KUKA KRL program: MyProgram_002().src

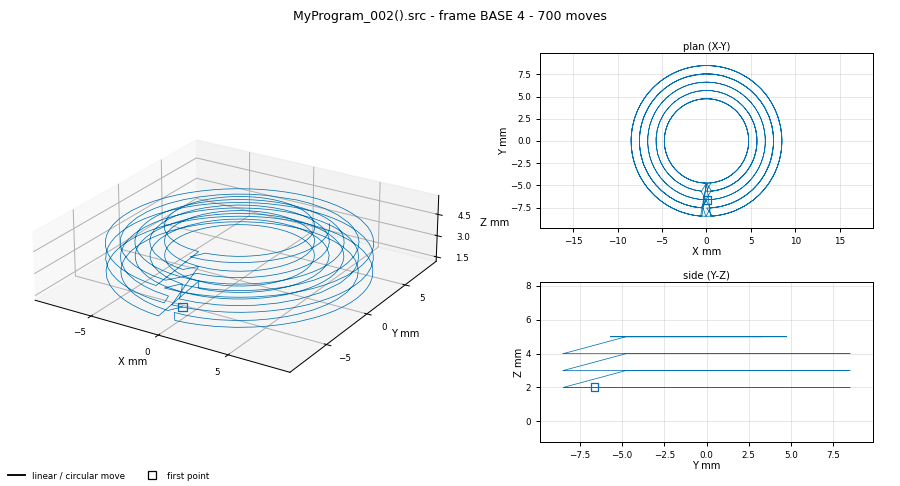
[picture p0: tool path of MyProgram_002().src in frame BASE 4, 700 of 700 moves have a stored position in this frame; points joined in program order, loops and branches not executed]
&ACCESS RVP
&REL 1
&PARAM TEMPLATE = C:\KRC\Roboter\Template\vorgabe
&PARAM EDITMASK = *
DEF MyProgram_002()
; ---- Setting reference (Base) ----
$BASE = BASE_DATA[4]

; --------------------------
; ---- Setting tool (TCP) ----
$TOOL = TOOL_DATA[3]
; --------------------------

$VEL.CP = VEL_APROX_PRINT
Startdeposition()
$VEL.CP = VEL_PRINT
LIN {X 0.0178,Y -6.6224,Z 2,A -3.1111,B 0,C 0,E1 0.1598,E2 90.0714} C_DIS
Enddeposition()
LIN {X 0.0178,Y -6.6224,Z 2,A -3.1111,B 0,C 0,E1 0.1598,E2 90.0714} C_DIS
Startdeposition()
$VEL.CP = VEL_PRINT
LIN {X -0.4593,Y -7.5388,Z 2,A -3.167,B 0,C 0,E1 0.1598,E2 90.0708} C_DIS
LIN {X -1.4599,Y -7.4149,Z 2,A -3.199,B 0,C 0,E1 0.1598,E2 90.0713} C_DIS
LIN {X -2.4674,Y -7.1388,Z 2,A -3.2242,B 0,C 0,E1 0.1598,E2 90.0713} C_DIS
LIN {X -3.4306,Y -6.7344,Z 2,A -3.2424,B 0,C 0,E1 0.1598,E2 90.0711} C_DIS
LIN {X -4.2642,Y -6.2384,Z 2,A -3.252,B 0,C 0,E1 0.1598,E2 90.0711} C_DIS
LIN {X -5.1322,Y -5.543,Z 2,A -3.2544,B 0,C 0,E1 0.1598,E2 90.071} C_DIS
LIN {X -5.6941,Y -4.9627,Z 2,A -3.2507,B 0,C 0,E1 0.1598,E2 90.071} C_DIS
LIN {X -6.1903,Y -4.3255,Z 2,A -3.242,B 0,C 0,E1 0.1598,E2 90.071} C_DIS
LIN {X -6.7788,Y -3.3392,Z 2,A -3.2218,B 0,C 0,E1 0.1598,E2 90.0708} C_DIS
LIN {X -7.1266,Y -2.5145,Z 2,A -3.2,B 0,C 0,E1 0.1598,E2 90.0708} C_DIS
LIN {X -7.4318,Y -1.3786,Z 2,A -3.1631,B 0,C 0,E1 0.1598,E2 90.0708} C_DIS
LIN {X -7.5532,Y -0.2507,Z 2,A -3.1202,B 0,C 0,E1 0.1598,E2 90.0708} C_DIS
LIN {X -7.507,Y 0.8388,Z 2,A -3.0728,B 0,C 0,E1 0.1598,E2 90.0709} C_DIS
LIN {X -7.3592,Y 1.6986,Z 2,A -3.0313,B 0,C 0,E1 0.1598,E2 90.0712} C_DIS
LIN {X -7.0429,Y 2.7423,Z 2,A -2.9756,B 0,C 0,E1 0.1598,E2 90.071} C_DIS
LIN {X -6.514,Y 3.8232,Z 2,A -2.9107,B 0,C 0,E1 0.1598,E2 90.0711} C_DIS
LIN {X -6.0604,Y 4.5077,Z 2,A -2.8655,B 0,C 0,E1 0.1598,E2 90.0715} C_DIS
LIN {X -5.5355,Y 5.1393,Z 2,A -2.8197,B 0,C 0,E1 0.1598,E2 90.0716} C_DIS
LIN {X -4.7193,Y 5.9031,Z 2,A -2.7574,B 0,C 0,E1 0.1598,E2 90.0716} C_DIS
LIN {X -3.7399,Y 6.5671,Z 2,A -2.6934,B 0,C 0,E1 0.1598,E2 90.0718} C_DIS
LIN {X -2.7889,Y 7.019,Z 2,A -2.6394,B 0,C 0,E1 0.1598,E2 90.072} C_DIS
LIN {X -1.9903,Y 7.2868,Z 2,A -2.5987,B 0,C 0,E1 0.1598,E2 90.072} C_DIS
LIN {X -1.1667,Y 7.463,Z 2,A -2.5609,B 0,C 0,E1 0.1598,E2 90.0721} C_DIS
LIN {X -0.118,Y 7.5562,Z 2,A -2.5182,B 0,C 0,E1 0.1598,E2 90.0722} C_DIS
LIN {X 1.0472,Y 7.4801,Z 2,A -2.4784,B 0,C 0,E1 0.1598,E2 90.0722} C_DIS
LIN {X 1.8826,Y 7.3157,Z 2,A -2.4545,B 0,C 0,E1 0.1598,E2 90.0722} C_DIS
LIN {X 2.9847,Y 6.9422,Z 2,A -2.4295,B 0,C 0,E1 0.1598,E2 90.0722} C_DIS
LIN {X 3.8476,Y 6.5002,Z 2,A -2.4163,B 0,C 0,E1 0.1598,E2 90.0722} C_DIS
LIN {X 4.7671,Y 5.8658,Z 2,A -2.409,B 0,C 0,E1 0.1598,E2 90.0722} C_DIS
LIN {X 5.5879,Y 5.0811,Z 2,A -2.4118,B 0,C 0,E1 0.1598,E2 90.072} C_DIS
LIN {X 6.1162,Y 4.4317,Z 2,A -2.4199,B 0,C 0,E1 0.1598,E2 90.072} C_DIS
LIN {X 6.5685,Y 3.7273,Z 2,A -2.433,B 0,C 0,E1 0.1598,E2 90.072} C_DIS
LIN {X 7.0263,Y 2.7862,Z 2,A -2.4557,B 0,C 0,E1 0.1598,E2 90.0717} C_DIS
LIN {X 7.3641,Y 1.6742,Z 2,A -2.4903,B 0,C 0,E1 0.1598,E2 90.0715} C_DIS
LIN {X 7.5359,Y 0.5664,Z 2,A -2.5309,B 0,C 0,E1 0.1598,E2 90.0715} C_DIS
LIN {X 7.5261,Y -0.6981,Z 2,A -2.5848,B 0,C 0,E1 0.1598,E2 90.0713} C_DIS
LIN {X 7.3558,Y -1.7123,Z 2,A -2.6343,B 0,C 0,E1 0.1598,E2 90.0715} C_DIS
LIN {X 7.0595,Y -2.6971,Z 2,A -2.6869,B 0,C 0,E1 0.1598,E2 90.0714} C_DIS
LIN {X 6.5954,Y -3.6789,Z 2,A -2.7457,B 0,C 0,E1 0.1598,E2 90.0714} C_DIS
LIN {X 6.1284,Y -4.4233,Z 2,A -2.7946,B 0,C 0,E1 0.1598,E2 90.0715} C_DIS
LIN {X 5.3883,Y -5.2916,Z 2,A -2.8585,B 0,C 0,E1 0.1598,E2 90.0714} C_DIS
LIN {X 4.762,Y -5.8618,Z 2,A -2.9059,B 0,C 0,E1 0.1598,E2 90.0715} C_DIS
LIN {X 3.8982,Y -6.4739,Z 2,A -2.9635,B 0,C 0,E1 0.1598,E2 90.0715} C_DIS
LIN {X 2.7755,Y -7.0305,Z 2,A -3.0283,B 0,C 0,E1 0.1598,E2 90.0714} C_DIS
LIN {X 1.7367,Y -7.3513,Z 2,A -3.0801,B 0,C 0,E1 0.1598,E2 90.0714} C_DIS
LIN {X 0.7907,Y -7.5156,Z 2,A -3.1218,B 0,C 0,E1 0.1598,E2 90.0714} C_DIS
LIN {X 0.024,Y -7.5549,Z 2,A -3.1516,B 0,C 0,E1 0.1598,E2 90.0714} C_DIS
Enddeposition()
LIN {X 0.024,Y -7.5549,Z 2,A -3.1516,B 0,C 0,E1 0.1598,E2 90.0714} C_DIS
Startdeposition()
$VEL.CP = VEL_PRINT
LIN {X 0.6615,Y -8.4625,Z 2,A -3.1663,B 0,C 0,E1 0.1598,E2 90.0708} C_DIS
LIN {X 1.4734,Y -8.3591,Z 2,A -3.1326,B 0,C 0,E1 0.1598,E2 90.0714} C_DIS
LIN {X 2.2716,Y -8.1784,Z 2,A -3.0957,B 0,C 0,E1 0.1598,E2 90.0714} C_DIS
LIN {X 3.2398,Y -7.8482,Z 2,A -3.0462,B 0,C 0,E1 0.1598,E2 90.0714} C_DIS
LIN {X 4.3203,Y -7.3105,Z 2,A -2.9837,B 0,C 0,E1 0.1598,E2 90.0714} C_DIS
LIN {X 5.1942,Y -6.7139,Z 2,A -2.9263,B 0,C 0,E1 0.1598,E2 90.0715} C_DIS
LIN {X 5.8372,Y -6.1633,Z 2,A -2.8794,B 0,C 0,E1 0.1598,E2 90.0715} C_DIS
LIN {X 6.4222,Y -5.5514,Z 2,A -2.8319,B 0,C 0,E1 0.1598,E2 90.0716} C_DIS
LIN {X 7.0647,Y -4.7107,Z 2,A -2.7724,B 0,C 0,E1 0.1598,E2 90.0715} C_DIS
LIN {X 7.6515,Y -3.6709,Z 2,A -2.7066,B 0,C 0,E1 0.1598,E2 90.0715} C_DIS
LIN {X 7.9615,Y -2.9397,Z 2,A -2.6644,B 0,C 0,E1 0.1598,E2 90.0717} C_DIS
LIN {X 8.2023,Y -2.1829,Z 2,A -2.6234,B 0,C 0,E1 0.1598,E2 90.0717} C_DIS
LIN {X 8.3716,Y -1.4069,Z 2,A -2.5843,B 0,C 0,E1 0.1598,E2 90.0718} C_DIS
LIN {X 8.4662,Y -0.6183,Z 2,A -2.5473,B 0,C 0,E1 0.1598,E2 90.0718} C_DIS
LIN {X 8.4863,Y 0.1757,Z 2,A -2.5129,B 0,C 0,E1 0.1598,E2 90.0718} C_DIS
LIN {X 8.4313,Y 0.968,Z 2,A -2.4813,B 0,C 0,E1 0.1598,E2 90.0719} C_DIS
LIN {X 8.3033,Y 1.7517,Z 2,A -2.4527,B 0,C 0,E1 0.1598,E2 90.0719} C_DIS
LIN {X 8.1033,Y 2.5202,Z 2,A -2.4275,B 0,C 0,E1 0.1598,E2 90.0719} C_DIS
LIN {X 7.7584,Y 3.4511,Z 2,A -2.4005,B 0,C 0,E1 0.1598,E2 90.0719} C_DIS
LIN {X 7.165,Y 4.5511,Z 2,A -2.3757,B 0,C 0,E1 0.1598,E2 90.0717} C_DIS
LIN {X 6.6849,Y 5.2318,Z 2,A -2.365,B 0,C 0,E1 0.1598,E2 90.0721} C_DIS
LIN {X 6.1405,Y 5.8622,Z 2,A -2.3584,B 0,C 0,E1 0.1598,E2 90.0721} C_DIS
LIN {X 5.3784,Y 6.5716,Z 2,A -2.3564,B 0,C 0,E1 0.1598,E2 90.0721} C_DIS
LIN {X 4.6112,Y 7.1308,Z 2,A -2.3613,B 0,C 0,E1 0.1598,E2 90.0722} C_DIS
LIN {X 3.6186,Y 7.681,Z 2,A -2.3747,B 0,C 0,E1 0.1598,E2 90.0722} C_DIS
LIN {X 2.6506,Y 8.0636,Z 2,A -2.3944,B 0,C 0,E1 0.1598,E2 90.0722} C_DIS
LIN {X 1.8478,Y 8.2847,Z 2,A -2.4147,B 0,C 0,E1 0.1598,E2 90.0723} C_DIS
LIN {X 1.0272,Y 8.4264,Z 2,A -2.4391,B 0,C 0,E1 0.1598,E2 90.0723} C_DIS
LIN {X 0.1966,Y 8.4864,Z 2,A -2.4673,B 0,C 0,E1 0.1598,E2 90.0723} C_DIS
LIN {X -0.6357,Y 8.465,Z 2,A -2.4989,B 0,C 0,E1 0.1598,E2 90.0723} C_DIS
LIN {X -1.4619,Y 8.3604,Z 2,A -2.5338,B 0,C 0,E1 0.1598,E2 90.0722} C_DIS
LIN {X -2.2742,Y 8.1774,Z 2,A -2.5715,B 0,C 0,E1 0.1598,E2 90.0722} C_DIS
LIN {X -3.0645,Y 7.9151,Z 2,A -2.6117,B 0,C 0,E1 0.1598,E2 90.0721} C_DIS
LIN {X -3.8254,Y 7.5768,Z 2,A -2.654,B 0,C 0,E1 0.1598,E2 90.072} C_DIS
LIN {X -4.5496,Y 7.1657,Z 2,A -2.698,B 0,C 0,E1 0.1598,E2 90.0719} C_DIS
LIN {X -5.2302,Y 6.6859,Z 2,A -2.7433,B 0,C 0,E1 0.1598,E2 90.0719} C_DIS
LIN {X -5.8601,Y 6.1413,Z 2,A -2.7894,B 0,C 0,E1 0.1598,E2 90.0717} C_DIS
LIN {X -6.4342,Y 5.5382,Z 2,A -2.8359,B 0,C 0,E1 0.1598,E2 90.0717} C_DIS
LIN {X -6.9449,Y 4.8805,Z 2,A -2.8823,B 0,C 0,E1 0.1598,E2 90.0715} C_DIS
LIN {X -7.3896,Y 4.1765,Z 2,A -2.9282,B 0,C 0,E1 0.1598,E2 90.0715} C_DIS
LIN {X -7.763,Y 3.4322,Z 2,A -2.9732,B 0,C 0,E1 0.1598,E2 90.0713} C_DIS
LIN {X -8.062,Y 2.655,Z 2,A -3.0168,B 0,C 0,E1 0.1598,E2 90.0713} C_DIS
LIN {X -8.2835,Y 1.8523,Z 2,A -3.0587,B 0,C 0,E1 0.1598,E2 90.0712} C_DIS
LIN {X -8.4257,Y 1.0318,Z 2,A -3.0984,B 0,C 0,E1 0.1598,E2 90.0712} C_DIS
LIN {X -8.4869,Y 0.2014,Z 2,A -3.1355,B 0,C 0,E1 0.1598,E2 90.071} C_DIS
LIN {X -8.4655,Y -0.631,Z 2,A -3.1697,B 0,C 0,E1 0.1598,E2 90.071} C_DIS
LIN {X -8.3623,Y -1.4573,Z 2,A -3.2006,B 0,C 0,E1 0.1598,E2 90.071} C_DIS
LIN {X -8.1789,Y -2.2696,Z 2,A -3.2281,B 0,C 0,E1 0.1598,E2 90.071} C_DIS
LIN {X -7.9171,Y -3.0601,Z 2,A -3.2517,B 0,C 0,E1 0.1598,E2 90.071} C_DIS
LIN {X -7.5792,Y -3.8212,Z 2,A -3.2713,B 0,C 0,E1 0.1598,E2 90.071} C_DIS
LIN {X -7.0571,Y -4.7217,Z 2,A -3.2899,B 0,C 0,E1 0.1598,E2 90.0707} C_DIS
LIN {X -6.3174,Y -5.6752,Z 2,A -3.3028,B 0,C 0,E1 0.1598,E2 90.0707} C_DIS
LIN {X -5.5366,Y -6.4363,Z 2,A -3.3065,B 0,C 0,E1 0.1598,E2 90.0709} C_DIS
LIN {X -4.7817,Y -7.0119,Z 2,A -3.3032,B 0,C 0,E1 0.1598,E2 90.071} C_DIS
LIN {X -4.136,Y -7.4117,Z 2,A -3.2965,B 0,C 0,E1 0.1598,E2 90.071} C_DIS
LIN {X -3.4569,Y -7.7519,Z 2,A -3.286,B 0,C 0,E1 0.1598,E2 90.0711} C_DIS
LIN {X -2.7497,Y -8.0287,Z 2,A -3.2717,B 0,C 0,E1 0.1598,E2 90.0711} C_DIS
LIN {X -2.021,Y -8.2422,Z 2,A -3.2541,B 0,C 0,E1 0.1598,E2 90.0712} C_DIS
LIN {X -1.2762,Y -8.3903,Z 2,A -3.233,B 0,C 0,E1 0.1598,E2 90.0712} C_DIS
LIN {X -0.5212,Y -8.4723,Z 2,A -3.2088,B 0,C 0,E1 0.1598,E2 90.0712} C_DIS
LIN {X -0.5212,Y -8.4723,Z 2,A -3.2088,B 0,C 0,E1 0.1598,E2 90.0712} C_DIS
Enddeposition()
LIN {X 0.0002,Y -4.757,Z 3,A -3.0171,B 0,C 0,E1 0.1598,E2 90.0603} C_DIS
Startdeposition()
$VEL.CP = VEL_PRINT
LIN {X 0.0002,Y -4.757,Z 3,A -3.0228,B 0,C 0,E1 0.1598,E2 90.066} C_DIS
LIN {X -0.6823,Y -4.7037,Z 3,A -3.0504,B 0,C 0,E1 0.1598,E2 90.0709} C_DIS
LIN {X -1.2189,Y -4.5944,Z 3,A -3.0661,B 0,C 0,E1 0.1598,E2 90.0714} C_DIS
LIN {X -1.7393,Y -4.4237,Z 3,A -3.078,B 0,C 0,E1 0.1598,E2 90.0714} C_DIS
LIN {X -2.2363,Y -4.1936,Z 3,A -3.0865,B 0,C 0,E1 0.1598,E2 90.0714} C_DIS
LIN {X -2.7046,Y -3.9096,Z 3,A -3.0917,B 0,C 0,E1 0.1598,E2 90.0714} C_DIS
LIN {X -3.1363,Y -3.5726,Z 3,A -3.0933,B 0,C 0,E1 0.1598,E2 90.0714} C_DIS
LIN {X -3.5248,Y -3.1869,Z 3,A -3.0913,B 0,C 0,E1 0.1598,E2 90.0714} C_DIS
LIN {X -3.868,Y -2.7601,Z 3,A -3.0859,B 0,C 0,E1 0.1598,E2 90.0714} C_DIS
LIN {X -4.1606,Y -2.297,Z 3,A -3.0771,B 0,C 0,E1 0.1598,E2 90.0714} C_DIS
LIN {X -4.3949,Y -1.8023,Z 3,A -3.0649,B 0,C 0,E1 0.1598,E2 90.0714} C_DIS
LIN {X -4.5762,Y -1.2855,Z 3,A -3.0497,B 0,C 0,E1 0.1598,E2 90.0714} C_DIS
LIN {X -4.6927,Y -0.7504,Z 3,A -3.0315,B 0,C 0,E1 0.1598,E2 90.0714} C_DIS
LIN {X -4.7468,Y -0.2055,Z 3,A -3.0105,B 0,C 0,E1 0.1598,E2 90.0714} C_DIS
LIN {X -4.7423,Y 0.3421,Z 3,A -2.9873,B 0,C 0,E1 0.1598,E2 90.0714} C_DIS
LIN {X -4.6683,Y 0.8848,Z 3,A -2.9617,B 0,C 0,E1 0.1598,E2 90.0714} C_DIS
LIN {X -4.5367,Y 1.4164,Z 3,A -2.9345,B 0,C 0,E1 0.1598,E2 90.0715} C_DIS
LIN {X -4.3445,Y 1.9292,Z 3,A -2.9058,B 0,C 0,E1 0.1598,E2 90.0715} C_DIS
LIN {X -4.0931,Y 2.4158,Z 3,A -2.8761,B 0,C 0,E1 0.1598,E2 90.0716} C_DIS
LIN {X -3.7885,Y 2.8709,Z 3,A -2.8457,B 0,C 0,E1 0.1598,E2 90.0716} C_DIS
LIN {X -3.434,Y 3.2883,Z 3,A -2.8151,B 0,C 0,E1 0.1598,E2 90.0717} C_DIS
LIN {X -3.0321,Y 3.6604,Z 3,A -2.7846,B 0,C 0,E1 0.1598,E2 90.0717} C_DIS
LIN {X -2.5909,Y 3.9849,Z 3,A -2.7547,B 0,C 0,E1 0.1598,E2 90.0719} C_DIS
LIN {X -2.1155,Y 4.2567,Z 3,A -2.7257,B 0,C 0,E1 0.1598,E2 90.0719} C_DIS
LIN {X -1.6115,Y 4.4711,Z 3,A -2.6981,B 0,C 0,E1 0.1598,E2 90.0719} C_DIS
LIN {X -1.0866,Y 4.6274,Z 3,A -2.6722,B 0,C 0,E1 0.1598,E2 90.072} C_DIS
LIN {X -0.5471,Y 4.7215,Z 3,A -2.6483,B 0,C 0,E1 0.1598,E2 90.072} C_DIS
LIN {X -0.0003,Y 4.753,Z 3,A -2.6268,B 0,C 0,E1 0.1598,E2 90.072} C_DIS
LIN {X 0.5465,Y 4.7225,Z 3,A -2.608,B 0,C 0,E1 0.1598,E2 90.072} C_DIS
LIN {X 1.0858,Y 4.6272,Z 3,A -2.5921,B 0,C 0,E1 0.1598,E2 90.0721} C_DIS
LIN {X 1.6101,Y 4.469,Z 3,A -2.5794,B 0,C 0,E1 0.1598,E2 90.0721} C_DIS
LIN {X 2.1146,Y 4.2565,Z 3,A -2.5698,B 0,C 0,E1 0.1598,E2 90.0721} C_DIS
LIN {X 2.5892,Y 3.9833,Z 3,A -2.5638,B 0,C 0,E1 0.1598,E2 90.0721} C_DIS
LIN {X 3.0305,Y 3.6591,Z 3,A -2.5612,B 0,C 0,E1 0.1598,E2 90.0721} C_DIS
LIN {X 3.433,Y 3.2877,Z 3,A -2.5621,B 0,C 0,E1 0.1598,E2 90.0721} C_DIS
LIN {X 3.7883,Y 2.8711,Z 3,A -2.5666,B 0,C 0,E1 0.1598,E2 90.0721} C_DIS
LIN {X 4.0916,Y 2.4151,Z 3,A -2.5747,B 0,C 0,E1 0.1598,E2 90.0721} C_DIS
LIN {X 4.3444,Y 1.9293,Z 3,A -2.5859,B 0,C 0,E1 0.1598,E2 90.072} C_DIS
LIN {X 4.5367,Y 1.4166,Z 3,A -2.6005,B 0,C 0,E1 0.1598,E2 90.072} C_DIS
LIN {X 4.6699,Y 0.8853,Z 3,A -2.6181,B 0,C 0,E1 0.1598,E2 90.072} C_DIS
LIN {X 4.7423,Y 0.3424,Z 3,A -2.6384,B 0,C 0,E1 0.1598,E2 90.0719} C_DIS
LIN {X 4.7478,Y -0.2053,Z 3,A -2.6614,B 0,C 0,E1 0.1598,E2 90.0719} C_DIS
LIN {X 4.6939,Y -0.7501,Z 3,A -2.6864,B 0,C 0,E1 0.1598,E2 90.0719} C_DIS
LIN {X 4.5744,Y -1.2846,Z 3,A -2.7135,B 0,C 0,E1 0.1598,E2 90.0719} C_DIS
LIN {X 4.3976,Y -1.8028,Z 3,A -2.7419,B 0,C 0,E1 0.1598,E2 90.0718} C_DIS
LIN {X 4.1613,Y -2.2969,Z 3,A -2.7716,B 0,C 0,E1 0.1598,E2 90.0718} C_DIS
LIN {X 3.87,Y -2.7606,Z 3,A -2.8019,B 0,C 0,E1 0.1598,E2 90.0718} C_DIS
LIN {X 3.5258,Y -3.1866,Z 3,A -2.8326,B 0,C 0,E1 0.1598,E2 90.0718} C_DIS
LIN {X 3.1365,Y -3.5719,Z 3,A -2.8633,B 0,C 0,E1 0.1598,E2 90.0717} C_DIS
LIN {X 2.7044,Y -3.9081,Z 3,A -2.8934,B 0,C 0,E1 0.1598,E2 90.0717} C_DIS
LIN {X 2.2361,Y -4.1922,Z 3,A -2.9226,B 0,C 0,E1 0.1598,E2 90.0717} C_DIS
LIN {X 1.7398,Y -4.4234,Z 3,A -2.9507,B 0,C 0,E1 0.1598,E2 90.0717} C_DIS
LIN {X 1.2188,Y -4.5918,Z 3,A -2.9769,B 0,C 0,E1 0.1598,E2 90.0716} C_DIS
LIN {X 0.6827,Y -4.7037,Z 3,A -3.0014,B 0,C 0,E1 0.1598,E2 90.0716} C_DIS
LIN {X 0.0002,Y -4.757,Z 3,A -3.0287,B 0,C 0,E1 0.1598,E2 90.0716} C_DIS
Enddeposition()
LIN {X 0.0002,Y -4.757,Z 3,A -3.0287,B 0,C 0,E1 0.1598,E2 90.0716} C_DIS
Startdeposition()
$VEL.CP = VEL_PRINT
LIN {X 0.5659,Y -5.6547,Z 3,A -3.0454,B 0,C 0,E1 0.1598,E2 90.071} C_DIS
LIN {X 1.3547,Y -5.5195,Z 3,A -3.0113,B 0,C 0,E1 0.1598,E2 90.0715} C_DIS
LIN {X 2.1165,Y -5.2741,Z 3,A -2.9729,B 0,C 0,E1 0.1598,E2 90.0715} C_DIS
LIN {X 2.8372,Y -4.9256,Z 3,A -2.9317,B 0,C 0,E1 0.1598,E2 90.0716} C_DIS
LIN {X 3.5009,Y -4.4782,Z 3,A -2.8883,B 0,C 0,E1 0.1598,E2 90.0716} C_DIS
LIN {X 4.0958,Y -3.9425,Z 3,A -2.8437,B 0,C 0,E1 0.1598,E2 90.0716} C_DIS
LIN {X 4.6092,Y -3.3282,Z 3,A -2.7988,B 0,C 0,E1 0.1598,E2 90.0716} C_DIS
LIN {X 5.0292,Y -2.6467,Z 3,A -2.7544,B 0,C 0,E1 0.1598,E2 90.0716} C_DIS
LIN {X 5.3532,Y -1.9147,Z 3,A -2.7115,B 0,C 0,E1 0.1598,E2 90.0716} C_DIS
LIN {X 5.5679,Y -1.1434,Z 3,A -2.6708,B 0,C 0,E1 0.1598,E2 90.0716} C_DIS
LIN {X 5.6733,Y -0.35,Z 3,A -2.6333,B 0,C 0,E1 0.1598,E2 90.0717} C_DIS
LIN {X 5.6642,Y 0.4503,Z 3,A -2.5997,B 0,C 0,E1 0.1598,E2 90.0717} C_DIS
LIN {X 5.5458,Y 1.2418,Z 3,A -2.5706,B 0,C 0,E1 0.1598,E2 90.0717} C_DIS
LIN {X 5.3166,Y 2.0087,Z 3,A -2.5465,B 0,C 0,E1 0.1598,E2 90.0718} C_DIS
LIN {X 4.8879,Y 2.9128,Z 3,A -2.5239,B 0,C 0,E1 0.1598,E2 90.0717} C_DIS
LIN {X 4.2073,Y 3.8229,Z 3,A -2.5105,B 0,C 0,E1 0.1598,E2 90.0717} C_DIS
LIN {X 3.615,Y 4.3886,Z 3,A -2.5087,B 0,C 0,E1 0.1598,E2 90.072} C_DIS
LIN {X 2.9467,Y 4.8621,Z 3,A -2.5134,B 0,C 0,E1 0.1598,E2 90.072} C_DIS
LIN {X 2.2169,Y 5.2338,Z 3,A -2.5246,B 0,C 0,E1 0.1598,E2 90.0721} C_DIS
LIN {X 1.4422,Y 5.4988,Z 3,A -2.5421,B 0,C 0,E1 0.1598,E2 90.0721} C_DIS
LIN {X 0.6371,Y 5.6481,Z 3,A -2.5655,B 0,C 0,E1 0.1598,E2 90.0721} C_DIS
LIN {X -0.181,Y 5.68,Z 3,A -2.5944,B 0,C 0,E1 0.1598,E2 90.0721} C_DIS
LIN {X -0.9954,Y 5.5962,Z 3,A -2.6279,B 0,C 0,E1 0.1598,E2 90.0721} C_DIS
LIN {X -1.7885,Y 5.3936,Z 3,A -2.6657,B 0,C 0,E1 0.1598,E2 90.0721} C_DIS
LIN {X -2.9131,Y 4.8877,Z 3,A -2.7284,B 0,C 0,E1 0.1598,E2 90.0718} C_DIS
LIN {X -3.6482,Y 4.3607,Z 3,A -2.7777,B 0,C 0,E1 0.1598,E2 90.0718} C_DIS
LIN {X -4.2376,Y 3.7904,Z 3,A -2.8234,B 0,C 0,E1 0.1598,E2 90.0716} C_DIS
LIN {X -4.7386,Y 3.1413,Z 3,A -2.8691,B 0,C 0,E1 0.1598,E2 90.0716} C_DIS
LIN {X -5.2815,Y 2.117,Z 3,A -2.9319,B 0,C 0,E1 0.1598,E2 90.0712} C_DIS
LIN {X -5.5389,Y 1.2778,Z 3,A -2.9769,B 0,C 0,E1 0.1598,E2 90.0712} C_DIS
LIN {X -5.6863,Y 0.2165,Z 3,A -3.0267,B 0,C 0,E1 0.1598,E2 90.071} C_DIS
LIN {X -5.6319,Y -0.7558,Z 3,A -3.0658,B 0,C 0,E1 0.1598,E2 90.071} C_DIS
LIN {X -5.4764,Y -1.5191,Z 3,A -3.0923,B 0,C 0,E1 0.1598,E2 90.0711} C_DIS
LIN {X -5.2196,Y -2.2546,Z 3,A -3.1139,B 0,C 0,E1 0.1598,E2 90.0711} C_DIS
LIN {X -4.8609,Y -2.9464,Z 3,A -3.1299,B 0,C 0,E1 0.1598,E2 90.0711} C_DIS
LIN {X -4.4131,Y -3.5841,Z 3,A -3.1404,B 0,C 0,E1 0.1598,E2 90.0711} C_DIS
LIN {X -3.6555,Y -4.3598,Z 3,A -3.1452,B 0,C 0,E1 0.1598,E2 90.0711} C_DIS
LIN {X -2.8468,Y -4.9172,Z 3,A -3.1391,B 0,C 0,E1 0.1598,E2 90.0712} C_DIS
LIN {X -2.1425,Y -5.2653,Z 3,A -3.1281,B 0,C 0,E1 0.1598,E2 90.0713} C_DIS
LIN {X -1.3959,Y -5.5111,Z 3,A -3.1111,B 0,C 0,E1 0.1598,E2 90.0713} C_DIS
LIN {X -0.6227,Y -5.6519,Z 3,A -3.0887,B 0,C 0,E1 0.1598,E2 90.0714} C_DIS
LIN {X -0.6227,Y -5.6519,Z 3,A -3.0887,B 0,C 0,E1 0.1598,E2 90.0714} C_DIS
Enddeposition()
LIN {X -0.0547,Y -6.6238,Z 3,A -3.1079,B 0,C 0,E1 0.1598,E2 90.0703} C_DIS
Startdeposition()
$VEL.CP = VEL_PRINT
LIN {X -0.9403,Y -6.5528,Z 3,A -3.1385,B 0,C 0,E1 0.1598,E2 90.0713} C_DIS
LIN {X -1.6368,Y -6.4121,Z 3,A -3.1582,B 0,C 0,E1 0.1598,E2 90.0713} C_DIS
LIN {X -2.3151,Y -6.2004,Z 3,A -3.1741,B 0,C 0,E1 0.1598,E2 90.0713} C_DIS
LIN {X -2.9667,Y -5.9167,Z 3,A -3.186,B 0,C 0,E1 0.1598,E2 90.0713} C_DIS
LIN {X -3.5839,Y -5.5645,Z 3,A -3.1938,B 0,C 0,E1 0.1598,E2 90.0713} C_DIS
LIN {X -4.1606,Y -5.1494,Z 3,A -3.1974,B 0,C 0,E1 0.1598,E2 90.0713} C_DIS
LIN {X -4.6878,Y -4.6728,Z 3,A -3.1966,B 0,C 0,E1 0.1598,E2 90.0712} C_DIS
LIN {X -5.1627,Y -4.1443,Z 3,A -3.1917,B 0,C 0,E1 0.1598,E2 90.0712} C_DIS
LIN {X -5.5767,Y -3.5667,Z 3,A -3.1826,B 0,C 0,E1 0.1598,E2 90.0712} C_DIS
LIN {X -5.9281,Y -2.9489,Z 3,A -3.1694,B 0,C 0,E1 0.1598,E2 90.0712} C_DIS
LIN {X -6.2073,Y -2.2953,Z 3,A -3.1521,B 0,C 0,E1 0.1598,E2 90.0712} C_DIS
LIN {X -6.4184,Y -1.6168,Z 3,A -3.1313,B 0,C 0,E1 0.1598,E2 90.0712} C_DIS
LIN {X -6.555,Y -0.9194,Z 3,A -3.107,B 0,C 0,E1 0.1598,E2 90.0712} C_DIS
LIN {X -6.6162,Y -0.2115,Z 3,A -3.0794,B 0,C 0,E1 0.1598,E2 90.0712} C_DIS
LIN {X -6.6006,Y 0.499,Z 3,A -3.049,B 0,C 0,E1 0.1598,E2 90.0712} C_DIS
LIN {X -6.5101,Y 1.2038,Z 3,A -3.016,B 0,C 0,E1 0.1598,E2 90.0713} C_DIS
LIN {X -6.344,Y 1.8948,Z 3,A -2.9808,B 0,C 0,E1 0.1598,E2 90.0713} C_DIS
LIN {X -6.1053,Y 2.5642,Z 3,A -2.9439,B 0,C 0,E1 0.1598,E2 90.0714} C_DIS
LIN {X -5.7956,Y 3.2039,Z 3,A -2.9056,B 0,C 0,E1 0.1598,E2 90.0714} C_DIS
LIN {X -5.4182,Y 3.8062,Z 3,A -2.8664,B 0,C 0,E1 0.1598,E2 90.0716} C_DIS
LIN {X -4.9762,Y 4.3628,Z 3,A -2.8267,B 0,C 0,E1 0.1598,E2 90.0716} C_DIS
LIN {X -4.4816,Y 4.8729,Z 3,A -2.787,B 0,C 0,E1 0.1598,E2 90.0717} C_DIS
LIN {X -3.9323,Y 5.3238,Z 3,A -2.7478,B 0,C 0,E1 0.1598,E2 90.0718} C_DIS
LIN {X -3.3399,Y 5.7162,Z 3,A -2.7094,B 0,C 0,E1 0.1598,E2 90.0718} C_DIS
LIN {X -2.7081,Y 6.0415,Z 3,A -2.6725,B 0,C 0,E1 0.1598,E2 90.072} C_DIS
LIN {X -2.0452,Y 6.2975,Z 3,A -2.6372,B 0,C 0,E1 0.1598,E2 90.072} C_DIS
LIN {X -1.3586,Y 6.4813,Z 3,A -2.6042,B 0,C 0,E1 0.1598,E2 90.072} C_DIS
LIN {X -0.656,Y 6.5872,Z 3,A -2.5738,B 0,C 0,E1 0.1598,E2 90.0721} C_DIS
LIN {X 0.0541,Y 6.6202,Z 3,A -2.5462,B 0,C 0,E1 0.1598,E2 90.0721} C_DIS
LIN {X 0.7632,Y 6.5737,Z 3,A -2.522,B 0,C 0,E1 0.1598,E2 90.0722} C_DIS
LIN {X 1.464,Y 6.4567,Z 3,A -2.5011,B 0,C 0,E1 0.1598,E2 90.0722} C_DIS
LIN {X 2.1474,Y 6.2615,Z 3,A -2.4841,B 0,C 0,E1 0.1598,E2 90.0722} C_DIS
LIN {X 2.8066,Y 5.996,Z 3,A -2.4709,B 0,C 0,E1 0.1598,E2 90.0722} C_DIS
LIN {X 3.4331,Y 5.6604,Z 3,A -2.462,B 0,C 0,E1 0.1598,E2 90.0722} C_DIS
LIN {X 4.0186,Y 5.2577,Z 3,A -2.4574,B 0,C 0,E1 0.1598,E2 90.0722} C_DIS
LIN {X 4.5596,Y 4.797,Z 3,A -2.4569,B 0,C 0,E1 0.1598,E2 90.0722} C_DIS
LIN {X 5.0477,Y 4.2805,Z 3,A -2.4607,B 0,C 0,E1 0.1598,E2 90.0722} C_DIS
LIN {X 5.4781,Y 3.7151,Z 3,A -2.4687,B 0,C 0,E1 0.1598,E2 90.0721} C_DIS
LIN {X 5.8459,Y 3.1071,Z 3,A -2.4809,B 0,C 0,E1 0.1598,E2 90.0721} C_DIS
LIN {X 6.1454,Y 2.4627,Z 3,A -2.4971,B 0,C 0,E1 0.1598,E2 90.0721} C_DIS
LIN {X 6.4225,Y 1.6185,Z 3,A -2.5224,B 0,C 0,E1 0.1598,E2 90.0717} C_DIS
LIN {X 6.5883,Y 0.6389,Z 3,A -2.5577,B 0,C 0,E1 0.1598,E2 90.0717} C_DIS
LIN {X 6.6212,Y -0.0031,Z 3,A -2.584,B 0,C 0,E1 0.1598,E2 90.0719} C_DIS
LIN {X 6.5897,Y -0.6453,Z 3,A -2.6124,B 0,C 0,E1 0.1598,E2 90.0719} C_DIS
LIN {X 6.4963,Y -1.2814,Z 3,A -2.6428,B 0,C 0,E1 0.1598,E2 90.0719} C_DIS
LIN {X 6.3414,Y -1.9054,Z 3,A -2.675,B 0,C 0,E1 0.1598,E2 90.0718} C_DIS
LIN {X 6.1258,Y -2.5111,Z 3,A -2.7086,B 0,C 0,E1 0.1598,E2 90.0718} C_DIS
LIN {X 5.8535,Y -3.0936,Z 3,A -2.7433,B 0,C 0,E1 0.1598,E2 90.0718} C_DIS
LIN {X 5.5261,Y -3.6468,Z 3,A -2.7788,B 0,C 0,E1 0.1598,E2 90.0718} C_DIS
LIN {X 5.1461,Y -4.1653,Z 3,A -2.8148,B 0,C 0,E1 0.1598,E2 90.0717} C_DIS
LIN {X 4.7178,Y -4.6447,Z 3,A -2.8509,B 0,C 0,E1 0.1598,E2 90.0717} C_DIS
LIN {X 4.2445,Y -5.0797,Z 3,A -2.8867,B 0,C 0,E1 0.1598,E2 90.0717} C_DIS
LIN {X 3.731,Y -5.4666,Z 3,A -2.922,B 0,C 0,E1 0.1598,E2 90.0717} C_DIS
LIN {X 3.1845,Y -5.8051,Z 3,A -2.9564,B 0,C 0,E1 0.1598,E2 90.0716} C_DIS
LIN {X 2.6061,Y -6.0863,Z 3,A -2.9895,B 0,C 0,E1 0.1598,E2 90.0716} C_DIS
LIN {X 2.0038,Y -6.3109,Z 3,A -3.0212,B 0,C 0,E1 0.1598,E2 90.0716} C_DIS
LIN {X 1.3824,Y -6.4765,Z 3,A -3.051,B 0,C 0,E1 0.1598,E2 90.0715} C_DIS
LIN {X 0.7478,Y -6.58,Z 3,A -3.0787,B 0,C 0,E1 0.1598,E2 90.0715} C_DIS
LIN {X -0.0547,Y -6.6238,Z 3,A -3.1099,B 0,C 0,E1 0.1598,E2 90.0715} C_DIS
Enddeposition()
LIN {X -0.0547,Y -6.6238,Z 3,A -3.1099,B 0,C 0,E1 0.1598,E2 90.0715} C_DIS
Startdeposition()
$VEL.CP = VEL_PRINT
LIN {X 0.4023,Y -7.5467,Z 3,A -3.1319,B 0,C 0,E1 0.1598,E2 90.0709} C_DIS
LIN {X 1.5507,Y -7.3959,Z 3,A -3.0839,B 0,C 0,E1 0.1598,E2 90.0714} C_DIS
LIN {X 2.8446,Y -7.0017,Z 3,A -3.0197,B 0,C 0,E1 0.1598,E2 90.0714} C_DIS
LIN {X 3.674,Y -6.6033,Z 3,A -2.9724,B 0,C 0,E1 0.1598,E2 90.0715} C_DIS
LIN {X 4.7661,Y -5.8666,Z 3,A -2.9009,B 0,C 0,E1 0.1598,E2 90.0715} C_DIS
LIN {X 5.7819,Y -4.8637,Z 3,A -2.8206,B 0,C 0,E1 0.1598,E2 90.0711} C_DIS
LIN {X 6.5682,Y -3.7346,Z 3,A -2.7439,B 0,C 0,E1 0.1598,E2 90.0713} C_DIS
LIN {X 7.2298,Y -2.199,Z 3,A -2.6538,B 0,C 0,E1 0.1598,E2 90.0708} C_DIS
LIN {X 7.5512,Y -0.3347,Z 3,A -2.5621,B 0,C 0,E1 0.1598,E2 90.0701} C_DIS
LIN {X 7.5512,Y -0.3347,Z 3,A -2.5631,B 0,C 0,E1 0.1598,E2 90.0712} C_DIS
LIN {X 7.4884,Y 1.0278,Z 3,A -2.5075,B 0,C 0,E1 0.1598,E2 90.071} C_DIS
LIN {X 7.2603,Y 2.0809,Z 3,A -2.4718,B 0,C 0,E1 0.1598,E2 90.0717} C_DIS
LIN {X 6.9759,Y 2.8946,Z 3,A -2.448,B 0,C 0,E1 0.1598,E2 90.0719} C_DIS
LIN {X 6.5993,Y 3.6698,Z 3,A -2.4291,B 0,C 0,E1 0.1598,E2 90.0719} C_DIS
LIN {X 6.1396,Y 4.3989,Z 3,A -2.4152,B 0,C 0,E1 0.1598,E2 90.072} C_DIS
LIN {X 5.5983,Y 5.0697,Z 3,A -2.4068,B 0,C 0,E1 0.1598,E2 90.072} C_DIS
LIN {X 4.7669,Y 5.866,Z 3,A -2.4037,B 0,C 0,E1 0.1598,E2 90.072} C_DIS
LIN {X 4.1157,Y 6.3395,Z 3,A -2.4079,B 0,C 0,E1 0.1598,E2 90.0722} C_DIS
LIN {X 3.1669,Y 6.858,Z 3,A -2.421,B 0,C 0,E1 0.1598,E2 90.0722} C_DIS
LIN {X 2.4787,Y 7.1348,Z 3,A -2.4348,B 0,C 0,E1 0.1598,E2 90.0722} C_DIS
LIN {X 1.7667,Y 7.343,Z 3,A -2.4523,B 0,C 0,E1 0.1598,E2 90.0722} C_DIS
LIN {X 0.8542,Y 7.5084,Z 3,A -2.4791,B 0,C 0,E1 0.1598,E2 90.0722} C_DIS
LIN {X -0.2995,Y 7.5462,Z 3,A -2.5201,B 0,C 0,E1 0.1598,E2 90.0722} C_DIS
LIN {X -1.1599,Y 7.4629,Z 3,A -2.5554,B 0,C 0,E1 0.1598,E2 90.0722} C_DIS
LIN {X -2.005,Y 7.2813,Z 3,A -2.5942,B 0,C 0,E1 0.1598,E2 90.0722} C_DIS
LIN {X -3.0251,Y 6.925,Z 3,A -2.6468,B 0,C 0,E1 0.1598,E2 90.072} C_DIS
LIN {X -4.0581,Y 6.3751,Z 3,A -2.708,B 0,C 0,E1 0.1598,E2 90.0718} C_DIS
LIN {X -4.7583,Y 5.8729,Z 3,A -2.755,B 0,C 0,E1 0.1598,E2 90.0718} C_DIS
LIN {X -5.5665,Y 5.1053,Z 3,A -2.8169,B 0,C 0,E1 0.1598,E2 90.0715} C_DIS
LIN {X -6.0209,Y 4.5596,Z 3,A -2.8567,B 0,C 0,E1 0.1598,E2 90.0716} C_DIS
LIN {X -6.4241,Y 3.9753,Z 3,A -2.8961,B 0,C 0,E1 0.1598,E2 90.0716} C_DIS
LIN {X -6.9273,Y 3.0196,Z 3,A -2.9546,B 0,C 0,E1 0.1598,E2 90.0712} C_DIS
LIN {X -7.2743,Y 2.0281,Z 3,A -3.009,B 0,C 0,E1 0.1598,E2 90.0712} C_DIS
LIN {X -7.4552,Y 1.2074,Z 3,A -3.0503,B 0,C 0,E1 0.1598,E2 90.0712} C_DIS
LIN {X -7.5445,Y 0.3717,Z 3,A -3.0887,B 0,C 0,E1 0.1598,E2 90.0712} C_DIS
LIN {X -7.5159,Y -0.7883,Z 3,A -3.1361,B 0,C 0,E1 0.1598,E2 90.0708} C_DIS
LIN {X -7.3438,Y -1.7653,Z 3,A -3.1711,B 0,C 0,E1 0.1598,E2 90.0709} C_DIS
LIN {X -7.0533,Y -2.7139,Z 3,A -3.2002,B 0,C 0,E1 0.1598,E2 90.0708} C_DIS
LIN {X -6.6068,Y -3.6627,Z 3,A -3.2238,B 0,C 0,E1 0.1598,E2 90.0708} C_DIS
LIN {X -6.229,Y -4.2694,Z 3,A -3.2358,B 0,C 0,E1 0.1598,E2 90.0711} C_DIS
LIN {X -5.6854,Y -4.9782,Z 3,A -3.2456,B 0,C 0,E1 0.1598,E2 90.0709} C_DIS
LIN {X -4.8305,Y -5.8077,Z 3,A -3.2491,B 0,C 0,E1 0.1598,E2 90.0709} C_DIS
LIN {X -4.2617,Y -6.2401,Z 3,A -3.2467,B 0,C 0,E1 0.1598,E2 90.0711} C_DIS
LIN {X -3.4291,Y -6.7351,Z 3,A -3.2371,B 0,C 0,E1 0.1598,E2 90.0711} C_DIS
LIN {X -2.4771,Y -7.1353,Z 3,A -3.2191,B 0,C 0,E1 0.1598,E2 90.0711} C_DIS
LIN {X -1.4818,Y -7.4104,Z 3,A -3.1942,B 0,C 0,E1 0.1598,E2 90.0713} C_DIS
LIN {X -0.3878,Y -7.5478,Z 3,A -3.16,B 0,C 0,E1 0.1598,E2 90.0713} C_DIS
LIN {X -0.3878,Y -7.5478,Z 3,A -3.16,B 0,C 0,E1 0.1598,E2 90.0713} C_DIS
Enddeposition()
LIN {X -0.075,Y -8.4864,Z 3,A -3.1873,B 0,C 0,E1 0.1598,E2 90.0702} C_DIS
Startdeposition()
$VEL.CP = VEL_PRINT
LIN {X -1.0165,Y -8.4281,Z 3,A -3.2204,B 0,C 0,E1 0.1598,E2 90.0712} C_DIS
LIN {X -1.7609,Y -8.3037,Z 3,A -3.2425,B 0,C 0,E1 0.1598,E2 90.0712} C_DIS
LIN {X -2.8343,Y -8.0038,Z 3,A -3.2691,B 0,C 0,E1 0.1598,E2 90.0712} C_DIS
LIN {X -3.763,Y -7.6075,Z 3,A -3.2864,B 0,C 0,E1 0.1598,E2 90.0712} C_DIS
LIN {X -4.4691,Y -7.2153,Z 3,A -3.2957,B 0,C 0,E1 0.1598,E2 90.0711} C_DIS
LIN {X -5.134,Y -6.7567,Z 3,A -3.3007,B 0,C 0,E1 0.1598,E2 90.0711} C_DIS
LIN {X -5.903,Y -6.1025,Z 3,A -3.3012,B 0,C 0,E1 0.1598,E2 90.0709} C_DIS
LIN {X -6.7522,Y -5.1469,Z 3,A -3.2918,B 0,C 0,E1 0.1598,E2 90.0706} C_DIS
LIN {X -7.377,Y -4.1982,Z 3,A -3.2749,B 0,C 0,E1 0.1598,E2 90.0706} C_DIS
LIN {X -7.7481,Y -3.4649,Z 3,A -3.2578,B 0,C 0,E1 0.1598,E2 90.0709} C_DIS
LIN {X -8.0466,Y -2.6992,Z 3,A -3.2366,B 0,C 0,E1 0.1598,E2 90.0709} C_DIS
LIN {X -8.2699,Y -1.9083,Z 3,A -3.2115,B 0,C 0,E1 0.1598,E2 90.0709} C_DIS
LIN {X -8.4159,Y -1.0995,Z 3,A -3.1828,B 0,C 0,E1 0.1598,E2 90.0709} C_DIS
LIN {X -8.4834,Y -0.2805,Z 3,A -3.1509,B 0,C 0,E1 0.1598,E2 90.071} C_DIS
LIN {X -8.4714,Y 0.5412,Z 3,A -3.1159,B 0,C 0,E1 0.1598,E2 90.071} C_DIS
LIN {X -8.3475,Y 1.561,Z 3,A -3.0682,B 0,C 0,E1 0.1598,E2 90.0709} C_DIS
LIN {X -8.0629,Y 2.6526,Z 3,A -3.0118,B 0,C 0,E1 0.1598,E2 90.0709} C_DIS
LIN {X -7.6795,Y 3.6218,Z 3,A -2.957,B 0,C 0,E1 0.1598,E2 90.0711} C_DIS
LIN {X -7.0961,Y 4.6546,Z 3,A -2.8922,B 0,C 0,E1 0.1598,E2 90.0711} C_DIS
LIN {X -6.6207,Y 5.3104,Z 3,A -2.8474,B 0,C 0,E1 0.1598,E2 90.0716} C_DIS
LIN {X -6.0847,Y 5.9177,Z 3,A -2.8021,B 0,C 0,E1 0.1598,E2 90.0716} C_DIS
LIN {X -5.4927,Y 6.4705,Z 3,A -2.7571,B 0,C 0,E1 0.1598,E2 90.0717} C_DIS
LIN {X -4.8506,Y 6.9644,Z 3,A -2.7127,B 0,C 0,E1 0.1598,E2 90.0718} C_DIS
LIN {X -4.1645,Y 7.3952,Z 3,A -2.6692,B 0,C 0,E1 0.1598,E2 90.0719} C_DIS
LIN {X -3.4406,Y 7.7589,Z 3,A -2.6272,B 0,C 0,E1 0.1598,E2 90.072} C_DIS
LIN {X -2.6852,Y 8.0519,Z 3,A -2.587,B 0,C 0,E1 0.1598,E2 90.072} C_DIS
LIN {X -1.9052,Y 8.2709,Z 3,A -2.549,B 0,C 0,E1 0.1598,E2 90.0722} C_DIS
LIN {X -1.1079,Y 8.4148,Z 3,A -2.5135,B 0,C 0,E1 0.1598,E2 90.0722} C_DIS
LIN {X -0.3007,Y 8.4825,Z 3,A -2.4809,B 0,C 0,E1 0.1598,E2 90.0722} C_DIS
LIN {X 0.5093,Y 8.4727,Z 3,A -2.4514,B 0,C 0,E1 0.1598,E2 90.0723} C_DIS
LIN {X 1.3145,Y 8.3844,Z 3,A -2.4253,B 0,C 0,E1 0.1598,E2 90.0723} C_DIS
LIN {X 2.1077,Y 8.2203,Z 3,A -2.4029,B 0,C 0,E1 0.1598,E2 90.0723} C_DIS
LIN {X 2.8817,Y 7.9816,Z 3,A -2.3844,B 0,C 0,E1 0.1598,E2 90.0723} C_DIS
LIN {X 3.6295,Y 7.6705,Z 3,A -2.3699,B 0,C 0,E1 0.1598,E2 90.0723} C_DIS
LIN {X 4.5194,Y 7.1875,Z 3,A -2.3574,B 0,C 0,E1 0.1598,E2 90.0723} C_DIS
LIN {X 5.3748,Y 6.5747,Z 3,A -2.3516,B 0,C 0,E1 0.1598,E2 90.0723} C_DIS
LIN {X 6.146,Y 5.856,Z 3,A -2.3535,B 0,C 0,E1 0.1598,E2 90.0721} C_DIS
LIN {X 6.696,Y 5.2166,Z 3,A -2.3603,B 0,C 0,E1 0.1598,E2 90.0721} C_DIS
LIN {X 7.18,Y 4.5259,Z 3,A -2.3717,B 0,C 0,E1 0.1598,E2 90.0721} C_DIS
LIN {X 7.5933,Y 3.7907,Z 3,A -2.3876,B 0,C 0,E1 0.1598,E2 90.0721} C_DIS
LIN {X 8.0084,Y 2.8217,Z 3,A -2.413,B 0,C 0,E1 0.1598,E2 90.0717} C_DIS
LIN {X 8.3238,Y 1.675,Z 3,A -2.4499,B 0,C 0,E1 0.1598,E2 90.0716} C_DIS
LIN {X 8.4636,Y 0.6503,Z 3,A -2.4884,B 0,C 0,E1 0.1598,E2 90.0717} C_DIS
LIN {X 8.486,Y -0.1767,Z 3,A -2.5228,B 0,C 0,E1 0.1598,E2 90.0718} C_DIS
LIN {X 8.4287,Y -1.002,Z 3,A -2.56,B 0,C 0,E1 0.1598,E2 90.0718} C_DIS
LIN {X 8.2914,Y -1.8179,Z 3,A -2.5997,B 0,C 0,E1 0.1598,E2 90.0718} C_DIS
LIN {X 8.0745,Y -2.6162,Z 3,A -2.6415,B 0,C 0,E1 0.1598,E2 90.0718} C_DIS
LIN {X 7.7812,Y -3.3899,Z 3,A -2.6852,B 0,C 0,E1 0.1598,E2 90.0717} C_DIS
LIN {X 7.4145,Y -4.1315,Z 3,A -2.7302,B 0,C 0,E1 0.1598,E2 90.0717} C_DIS
LIN {X 6.9775,Y -4.834,Z 3,A -2.7761,B 0,C 0,E1 0.1598,E2 90.0717} C_DIS
LIN {X 6.474,Y -5.4905,Z 3,A -2.8224,B 0,C 0,E1 0.1598,E2 90.0716} C_DIS
LIN {X 5.9085,Y -6.0943,Z 3,A -2.8688,B 0,C 0,E1 0.1598,E2 90.0716} C_DIS
LIN {X 5.2864,Y -6.6397,Z 3,A -2.9148,B 0,C 0,E1 0.1598,E2 90.0716} C_DIS
LIN {X 4.6146,Y -7.1225,Z 3,A -2.96,B 0,C 0,E1 0.1598,E2 90.0716} C_DIS
LIN {X 3.899,Y -7.5376,Z 3,A -3.0039,B 0,C 0,E1 0.1598,E2 90.0715} C_DIS
LIN {X 2.9549,Y -7.9594,Z 3,A -3.0564,B 0,C 0,E1 0.1598,E2 90.0715} C_DIS
LIN {X 1.9062,Y -8.2708,Z 3,A -3.108,B 0,C 0,E1 0.1598,E2 90.0714} C_DIS
LIN {X 1.1922,Y -8.4029,Z 3,A -3.1398,B 0,C 0,E1 0.1598,E2 90.0714} C_DIS
LIN {X 0.4695,Y -8.4745,Z 3,A -3.1694,B 0,C 0,E1 0.1598,E2 90.0714} C_DIS
LIN {X 0.4695,Y -8.4745,Z 3,A -3.1694,B 0,C 0,E1 0.1598,E2 90.0714} C_DIS
Enddeposition()
LIN {X 0.0002,Y -4.7527,Z 4,A -3.0137,B 0,C 0,E1 0.1598,E2 90.0604} C_DIS
Startdeposition()
$VEL.CP = VEL_PRINT
LIN {X 0.0002,Y -4.7527,Z 4,A -3.0193,B 0,C 0,E1 0.1598,E2 90.066} C_DIS
LIN {X 0.7986,Y -4.6829,Z 4,A -2.9919,B 0,C 0,E1 0.1598,E2 90.0709} C_DIS
LIN {X 1.4225,Y -4.5332,Z 4,A -2.9633,B 0,C 0,E1 0.1598,E2 90.0716} C_DIS
LIN {X 2.0204,Y -4.3006,Z 4,A -2.9315,B 0,C 0,E1 0.1598,E2 90.0716} C_DIS
LIN {X 2.5805,Y -3.988,Z 4,A -2.8976,B 0,C 0,E1 0.1598,E2 90.0716} C_DIS
LIN {X 3.0962,Y -3.6064,Z 4,A -2.8625,B 0,C 0,E1 0.1598,E2 90.0716} C_DIS
LIN {X 3.552,Y -3.1551,Z 4,A -2.8266,B 0,C 0,E1 0.1598,E2 90.0717} C_DIS
LIN {X 3.9442,Y -2.6476,Z 4,A -2.7907,B 0,C 0,E1 0.1598,E2 90.0717} C_DIS
LIN {X 4.2664,Y -2.0927,Z 4,A -2.7553,B 0,C 0,E1 0.1598,E2 90.0717} C_DIS
LIN {X 4.5072,Y -1.4981,Z 4,A -2.7212,B 0,C 0,E1 0.1598,E2 90.0717} C_DIS
LIN {X 4.6712,Y -0.8778,Z 4,A -2.6889,B 0,C 0,E1 0.1598,E2 90.0717} C_DIS
LIN {X 4.7457,Y -0.2406,Z 4,A -2.6592,B 0,C 0,E1 0.1598,E2 90.0718} C_DIS
LIN {X 4.7361,Y 0.4009,Z 4,A -2.6323,B 0,C 0,E1 0.1598,E2 90.0718} C_DIS
LIN {X 4.6365,Y 1.0349,Z 4,A -2.6092,B 0,C 0,E1 0.1598,E2 90.0718} C_DIS
LIN {X 4.4555,Y 1.6503,Z 4,A -2.5898,B 0,C 0,E1 0.1598,E2 90.0719} C_DIS
LIN {X 4.1919,Y 2.2351,Z 4,A -2.5748,B 0,C 0,E1 0.1598,E2 90.0719} C_DIS
LIN {X 3.8544,Y 2.7808,Z 4,A -2.5641,B 0,C 0,E1 0.1598,E2 90.0719} C_DIS
LIN {X 3.445,Y 3.2748,Z 4,A -2.5583,B 0,C 0,E1 0.1598,E2 90.072} C_DIS
LIN {X 2.9718,Y 3.7082,Z 4,A -2.5575,B 0,C 0,E1 0.1598,E2 90.072} C_DIS
LIN {X 2.4442,Y 4.0734,Z 4,A -2.5615,B 0,C 0,E1 0.1598,E2 90.072} C_DIS
LIN {X 1.8728,Y 4.3648,Z 4,A -2.5703,B 0,C 0,E1 0.1598,E2 90.072} C_DIS
LIN {X 1.2684,Y 4.5793,Z 4,A -2.5836,B 0,C 0,E1 0.1598,E2 90.072} C_DIS
LIN {X 0.6398,Y 4.7086,Z 4,A -2.6013,B 0,C 0,E1 0.1598,E2 90.072} C_DIS
LIN {X -0.0002,Y 4.7527,Z 4,A -2.6231,B 0,C 0,E1 0.1598,E2 90.072} C_DIS
LIN {X -0.6402,Y 4.7087,Z 4,A -2.6485,B 0,C 0,E1 0.1598,E2 90.072} C_DIS
LIN {X -1.2688,Y 4.5795,Z 4,A -2.6771,B 0,C 0,E1 0.1598,E2 90.072} C_DIS
LIN {X -1.8741,Y 4.3662,Z 4,A -2.7084,B 0,C 0,E1 0.1598,E2 90.072} C_DIS
LIN {X -2.445,Y 4.0738,Z 4,A -2.7418,B 0,C 0,E1 0.1598,E2 90.0719} C_DIS
LIN {X -2.9721,Y 3.7081,Z 4,A -2.7766,B 0,C 0,E1 0.1598,E2 90.0719} C_DIS
LIN {X -3.4439,Y 3.2733,Z 4,A -2.8123,B 0,C 0,E1 0.1598,E2 90.0717} C_DIS
LIN {X -3.8541,Y 2.7799,Z 4,A -2.8481,B 0,C 0,E1 0.1598,E2 90.0717} C_DIS
LIN {X -4.1937,Y 2.2356,Z 4,A -2.8835,B 0,C 0,E1 0.1598,E2 90.0716} C_DIS
LIN {X -4.4558,Y 1.6499,Z 4,A -2.9178,B 0,C 0,E1 0.1598,E2 90.0716} C_DIS
LIN {X -4.6366,Y 1.0344,Z 4,A -2.9504,B 0,C 0,E1 0.1598,E2 90.0714} C_DIS
LIN {X -4.7359,Y 0.4005,Z 4,A -2.9807,B 0,C 0,E1 0.1598,E2 90.0714} C_DIS
LIN {X -4.7455,Y -0.241,Z 4,A -3.0081,B 0,C 0,E1 0.1598,E2 90.0714} C_DIS
LIN {X -4.6697,Y -0.8779,Z 4,A -3.0321,B 0,C 0,E1 0.1598,E2 90.0714} C_DIS
LIN {X -4.5081,Y -1.4988,Z 4,A -3.0524,B 0,C 0,E1 0.1598,E2 90.0714} C_DIS
LIN {X -4.265,Y -2.0924,Z 4,A -3.0685,B 0,C 0,E1 0.1598,E2 90.0714} C_DIS
LIN {X -3.944,Y -2.6477,Z 4,A -3.0801,B 0,C 0,E1 0.1598,E2 90.0714} C_DIS
LIN {X -3.5533,Y -3.1566,Z 4,A -3.0872,B 0,C 0,E1 0.1598,E2 90.0714} C_DIS
LIN {X -3.0946,Y -3.6051,Z 4,A -3.0893,B 0,C 0,E1 0.1598,E2 90.0714} C_DIS
LIN {X -2.5804,Y -3.9885,Z 4,A -3.0866,B 0,C 0,E1 0.1598,E2 90.0714} C_DIS
LIN {X -2.02,Y -4.3006,Z 4,A -3.0793,B 0,C 0,E1 0.1598,E2 90.0714} C_DIS
LIN {X -1.422,Y -4.5329,Z 4,A -3.0671,B 0,C 0,E1 0.1598,E2 90.0714} C_DIS
LIN {X -0.7986,Y -4.6845,Z 4,A -3.0507,B 0,C 0,E1 0.1598,E2 90.0714} C_DIS
LIN {X 0.0002,Y -4.7527,Z 4,A -3.0242,B 0,C 0,E1 0.1598,E2 90.0715} C_DIS
Enddeposition()
LIN {X 0.0002,Y -4.7527,Z 4,A -3.0242,B 0,C 0,E1 0.1598,E2 90.0715} C_DIS
Startdeposition()
$VEL.CP = VEL_PRINT
LIN {X -0.5692,Y -5.6561,Z 4,A -3.0829,B 0,C 0,E1 0.1598,E2 90.0709} C_DIS
LIN {X -1.3093,Y -5.5324,Z 4,A -3.1054,B 0,C 0,E1 0.1598,E2 90.0714} C_DIS
LIN {X -2.2024,Y -5.2458,Z 4,A -3.126,B 0,C 0,E1 0.1598,E2 90.0714} C_DIS
LIN {X -3.4012,Y -4.5614,Z 4,A -3.1409,B 0,C 0,E1 0.1598,E2 90.0711} C_DIS
LIN {X -4.1629,Y -3.8681,Z 4,A -3.1397,B 0,C 0,E1 0.1598,E2 90.0711} C_DIS
LIN {X -4.6783,Y -3.2254,Z 4,A -3.1315,B 0,C 0,E1 0.1598,E2 90.0711} C_DIS
LIN {X -5.0967,Y -2.5155,Z 4,A -3.1169,B 0,C 0,E1 0.1598,E2 90.0711} C_DIS
LIN {X -5.4738,Y -1.5568,Z 4,A -3.0901,B 0,C 0,E1 0.1598,E2 90.0709} C_DIS
LIN {X -5.6694,Y -0.4229,Z 4,A -3.0494,B 0,C 0,E1 0.1598,E2 90.0709} C_DIS
LIN {X -5.6695,Y 0.392,Z 4,A -3.0154,B 0,C 0,E1 0.1598,E2 90.0712} C_DIS
LIN {X -5.5556,Y 1.1986,Z 4,A -2.9773,B 0,C 0,E1 0.1598,E2 90.0712} C_DIS
LIN {X -5.3263,Y 1.9804,Z 4,A -2.936,B 0,C 0,E1 0.1598,E2 90.0714} C_DIS
LIN {X -4.9914,Y 2.7232,Z 4,A -2.8924,B 0,C 0,E1 0.1598,E2 90.0714} C_DIS
LIN {X -4.6177,Y 3.3251,Z 4,A -2.8533,B 0,C 0,E1 0.1598,E2 90.0715} C_DIS
LIN {X -3.8698,Y 4.1709,Z 4,A -2.79,B 0,C 0,E1 0.1598,E2 90.0715} C_DIS
LIN {X -3.1009,Y 4.7656,Z 4,A -2.7368,B 0,C 0,E1 0.1598,E2 90.0718} C_DIS
LIN {X -2.4214,Y 5.1438,Z 4,A -2.6959,B 0,C 0,E1 0.1598,E2 90.0719} C_DIS
LIN {X -1.6962,Y 5.4244,Z 4,A -2.6574,B 0,C 0,E1 0.1598,E2 90.0719} C_DIS
LIN {X -0.9402,Y 5.6051,Z 4,A -2.6219,B 0,C 0,E1 0.1598,E2 90.0721} C_DIS
LIN {X -0.1665,Y 5.6797,Z 4,A -2.5902,B 0,C 0,E1 0.1598,E2 90.0721} C_DIS
LIN {X 0.6104,Y 5.652,Z 4,A -2.5627,B 0,C 0,E1 0.1598,E2 90.0721} C_DIS
LIN {X 1.3756,Y 5.5145,Z 4,A -2.5403,B 0,C 0,E1 0.1598,E2 90.0721} C_DIS
LIN {X 2.1159,Y 5.2768,Z 4,A -2.523,B 0,C 0,E1 0.1598,E2 90.0721} C_DIS
LIN {X 2.8159,Y 4.9385,Z 4,A -2.5114,B 0,C 0,E1 0.1598,E2 90.0721} C_DIS
LIN {X 3.4622,Y 4.5062,Z 4,A -2.5058,B 0,C 0,E1 0.1598,E2 90.0721} C_DIS
LIN {X 4.0447,Y 3.9916,Z 4,A -2.5061,B 0,C 0,E1 0.1598,E2 90.0721} C_DIS
LIN {X 4.5516,Y 3.4024,Z 4,A -2.5123,B 0,C 0,E1 0.1598,E2 90.0721} C_DIS
LIN {X 4.9741,Y 2.7498,Z 4,A -2.5243,B 0,C 0,E1 0.1598,E2 90.072} C_DIS
LIN {X 5.304,Y 2.0459,Z 4,A -2.5419,B 0,C 0,E1 0.1598,E2 90.072} C_DIS
LIN {X 5.5333,Y 1.303,Z 4,A -2.5649,B 0,C 0,E1 0.1598,E2 90.0718} C_DIS
LIN {X 5.6606,Y 0.5358,Z 4,A -2.5927,B 0,C 0,E1 0.1598,E2 90.0718} C_DIS
LIN {X 5.6784,Y -0.2415,Z 4,A -2.6249,B 0,C 0,E1 0.1598,E2 90.0718} C_DIS
LIN {X 5.5918,Y -1.014,Z 4,A -2.6609,B 0,C 0,E1 0.1598,E2 90.0718} C_DIS
LIN {X 5.4019,Y -1.7678,Z 4,A -2.6998,B 0,C 0,E1 0.1598,E2 90.0717} C_DIS
LIN {X 5.1105,Y -2.4886,Z 4,A -2.7411,B 0,C 0,E1 0.1598,E2 90.0717} C_DIS
LIN {X 4.7229,Y -3.1625,Z 4,A -2.7839,B 0,C 0,E1 0.1598,E2 90.0717} C_DIS
LIN {X 4.247,Y -3.7774,Z 4,A -2.8275,B 0,C 0,E1 0.1598,E2 90.0717} C_DIS
LIN {X 3.693,Y -4.323,Z 4,A -2.871,B 0,C 0,E1 0.1598,E2 90.0717} C_DIS
LIN {X 3.0685,Y -4.7862,Z 4,A -2.9136,B 0,C 0,E1 0.1598,E2 90.0716} C_DIS
LIN {X 2.3866,Y -5.1598,Z 4,A -2.9545,B 0,C 0,E1 0.1598,E2 90.0716} C_DIS
LIN {X 1.4743,Y -5.4953,Z 4,A -3.0022,B 0,C 0,E1 0.1598,E2 90.0716} C_DIS
LIN {X 0.4761,Y -5.665,Z 4,A -3.0461,B 0,C 0,E1 0.1598,E2 90.0716} C_DIS
LIN {X 0.4761,Y -5.665,Z 4,A -3.0461,B 0,C 0,E1 0.1598,E2 90.0716} C_DIS
Enddeposition()
LIN {X -0.0405,Y -6.6236,Z 4,A -3.1046,B 0,C 0,E1 0.1598,E2 90.0703} C_DIS
Startdeposition()
$VEL.CP = VEL_PRINT
LIN {X 0.8459,Y -6.5644,Z 4,A -3.0707,B 0,C 0,E1 0.1598,E2 90.0714} C_DIS
LIN {X 1.5451,Y -6.4377,Z 4,A -3.0397,B 0,C 0,E1 0.1598,E2 90.0715} C_DIS
LIN {X 2.2262,Y -6.235,Z 4,A -3.0061,B 0,C 0,E1 0.1598,E2 90.0715} C_DIS
LIN {X 2.8823,Y -5.9616,Z 4,A -2.9704,B 0,C 0,E1 0.1598,E2 90.0715} C_DIS
LIN {X 3.5046,Y -5.6183,Z 4,A -2.933,B 0,C 0,E1 0.1598,E2 90.0716} C_DIS
LIN {X 4.0855,Y -5.2087,Z 4,A -2.8943,B 0,C 0,E1 0.1598,E2 90.0716} C_DIS
LIN {X 4.6201,Y -4.7403,Z 4,A -2.8548,B 0,C 0,E1 0.1598,E2 90.0716} C_DIS
LIN {X 5.102,Y -4.2181,Z 4,A -2.815,B 0,C 0,E1 0.1598,E2 90.0716} C_DIS
LIN {X 5.5246,Y -3.6467,Z 4,A -2.7752,B 0,C 0,E1 0.1598,E2 90.0717} C_DIS
LIN {X 5.8839,Y -3.0334,Z 4,A -2.7359,B 0,C 0,E1 0.1598,E2 90.0717} C_DIS
LIN {X 6.1753,Y -2.3851,Z 4,A -2.6977,B 0,C 0,E1 0.1598,E2 90.0717} C_DIS
LIN {X 6.3949,Y -1.7093,Z 4,A -2.6609,B 0,C 0,E1 0.1598,E2 90.0717} C_DIS
LIN {X 6.542,Y -1.0139,Z 4,A -2.626,B 0,C 0,E1 0.1598,E2 90.0718} C_DIS
LIN {X 6.6125,Y -0.3069,Z 4,A -2.5934,B 0,C 0,E1 0.1598,E2 90.0718} C_DIS
LIN {X 6.607,Y 0.4038,Z 4,A -2.5635,B 0,C 0,E1 0.1598,E2 90.0718} C_DIS
LIN {X 6.5278,Y 1.1101,Z 4,A -2.5365,B 0,C 0,E1 0.1598,E2 90.0719} C_DIS
LIN {X 6.37,Y 1.803,Z 4,A -2.5129,B 0,C 0,E1 0.1598,E2 90.0719} C_DIS
LIN {X 6.1398,Y 2.4754,Z 4,A -2.4929,B 0,C 0,E1 0.1598,E2 90.0719} C_DIS
LIN {X 5.8383,Y 3.1188,Z 4,A -2.4768,B 0,C 0,E1 0.1598,E2 90.072} C_DIS
LIN {X 5.4696,Y 3.7263,Z 4,A -2.4647,B 0,C 0,E1 0.1598,E2 90.072} C_DIS
LIN {X 5.0416,Y 4.2937,Z 4,A -2.4565,B 0,C 0,E1 0.1598,E2 90.0721} C_DIS
LIN {X 4.5492,Y 4.8063,Z 4,A -2.453,B 0,C 0,E1 0.1598,E2 90.0721} C_DIS
LIN {X 4.0076,Y 5.2662,Z 4,A -2.4535,B 0,C 0,E1 0.1598,E2 90.0721} C_DIS
LIN {X 3.4211,Y 5.6675,Z 4,A -2.4582,B 0,C 0,E1 0.1598,E2 90.0721} C_DIS
LIN {X 2.7942,Y 6.0022,Z 4,A -2.4673,B 0,C 0,E1 0.1598,E2 90.0722} C_DIS
LIN {X 2.1343,Y 6.2657,Z 4,A -2.4805,B 0,C 0,E1 0.1598,E2 90.0722} C_DIS
LIN {X 1.4503,Y 6.4592,Z 4,A -2.4976,B 0,C 0,E1 0.1598,E2 90.0722} C_DIS
LIN {X 0.7497,Y 6.5789,Z 4,A -2.5184,B 0,C 0,E1 0.1598,E2 90.0722} C_DIS
LIN {X 0.0403,Y 6.6208,Z 4,A -2.5428,B 0,C 0,E1 0.1598,E2 90.0722} C_DIS
LIN {X -0.6696,Y 6.5871,Z 4,A -2.5705,B 0,C 0,E1 0.1598,E2 90.0722} C_DIS
LIN {X -1.3719,Y 6.4783,Z 4,A -2.601,B 0,C 0,E1 0.1598,E2 90.0722} C_DIS
LIN {X -2.0578,Y 6.2916,Z 4,A -2.6341,B 0,C 0,E1 0.1598,E2 90.072} C_DIS
LIN {X -2.7202,Y 6.0341,Z 4,A -2.6694,B 0,C 0,E1 0.1598,E2 90.072} C_DIS
LIN {X -3.3521,Y 5.7092,Z 4,A -2.7064,B 0,C 0,E1 0.1598,E2 90.072} C_DIS
LIN {X -3.9448,Y 5.3171,Z 4,A -2.7447,B 0,C 0,E1 0.1598,E2 90.0718} C_DIS
LIN {X -4.4919,Y 4.8635,Z 4,A -2.7839,B 0,C 0,E1 0.1598,E2 90.0718} C_DIS
LIN {X -4.9862,Y 4.353,Z 4,A -2.8236,B 0,C 0,E1 0.1598,E2 90.0717} C_DIS
LIN {X -5.4264,Y 3.795,Z 4,A -2.8633,B 0,C 0,E1 0.1598,E2 90.0717} C_DIS
LIN {X -5.8024,Y 3.1919,Z 4,A -2.9025,B 0,C 0,E1 0.1598,E2 90.0715} C_DIS
LIN {X -6.1101,Y 2.5512,Z 4,A -2.9408,B 0,C 0,E1 0.1598,E2 90.0715} C_DIS
LIN {X -6.3462,Y 1.8808,Z 4,A -2.9776,B 0,C 0,E1 0.1598,E2 90.0714} C_DIS
LIN {X -6.5103,Y 1.1894,Z 4,A -3.0127,B 0,C 0,E1 0.1598,E2 90.0714} C_DIS
LIN {X -6.6025,Y 0.4847,Z 4,A -3.0458,B 0,C 0,E1 0.1598,E2 90.0713} C_DIS
LIN {X -6.6173,Y -0.2258,Z 4,A -3.0762,B 0,C 0,E1 0.1598,E2 90.0713} C_DIS
LIN {X -6.5528,Y -0.9335,Z 4,A -3.1036,B 0,C 0,E1 0.1598,E2 90.0712} C_DIS
LIN {X -6.4151,Y -1.6307,Z 4,A -3.1279,B 0,C 0,E1 0.1598,E2 90.0712} C_DIS
LIN {X -6.2021,Y -2.3086,Z 4,A -3.1486,B 0,C 0,E1 0.1598,E2 90.0712} C_DIS
LIN {X -5.9215,Y -2.9616,Z 4,A -3.1658,B 0,C 0,E1 0.1598,E2 90.0712} C_DIS
LIN {X -5.569,Y -3.5788,Z 4,A -3.1789,B 0,C 0,E1 0.1598,E2 90.0712} C_DIS
LIN {X -5.1529,Y -4.1549,Z 4,A -3.1879,B 0,C 0,E1 0.1598,E2 90.0712} C_DIS
LIN {X -4.678,Y -4.6835,Z 4,A -3.1928,B 0,C 0,E1 0.1598,E2 90.0712} C_DIS
LIN {X -4.1491,Y -5.1582,Z 4,A -3.1934,B 0,C 0,E1 0.1598,E2 90.0712} C_DIS
LIN {X -3.5724,Y -5.5733,Z 4,A -3.1898,B 0,C 0,E1 0.1598,E2 90.0712} C_DIS
LIN {X -2.9545,Y -5.9245,Z 4,A -3.182,B 0,C 0,E1 0.1598,E2 90.0712} C_DIS
LIN {X -2.3027,Y -6.2078,Z 4,A -3.1701,B 0,C 0,E1 0.1598,E2 90.0713} C_DIS
LIN {X -1.6232,Y -6.4161,Z 4,A -3.154,B 0,C 0,E1 0.1598,E2 90.0713} C_DIS
LIN {X -0.926,Y -6.553,Z 4,A -3.1342,B 0,C 0,E1 0.1598,E2 90.0713} C_DIS
LIN {X -0.0405,Y -6.6236,Z 4,A -3.1047,B 0,C 0,E1 0.1598,E2 90.0714} C_DIS
Enddeposition()
LIN {X -0.0405,Y -6.6236,Z 4,A -3.1047,B 0,C 0,E1 0.1598,E2 90.0714} C_DIS
Startdeposition()
$VEL.CP = VEL_PRINT
LIN {X -0.6131,Y -7.5265,Z 4,A -3.1635,B 0,C 0,E1 0.1598,E2 90.0708} C_DIS
LIN {X -1.5721,Y -7.3914,Z 4,A -3.1935,B 0,C 0,E1 0.1598,E2 90.0713} C_DIS
LIN {X -2.4268,Y -7.1584,Z 4,A -3.215,B 0,C 0,E1 0.1598,E2 90.0713} C_DIS
LIN {X -3.3842,Y -6.757,Z 4,A -3.2331,B 0,C 0,E1 0.1598,E2 90.0712} C_DIS
LIN {X -4.2118,Y -6.2746,Z 4,A -3.243,B 0,C 0,E1 0.1598,E2 90.0711} C_DIS
LIN {X -5.0922,Y -5.5781,Z 4,A -3.2459,B 0,C 0,E1 0.1598,E2 90.0711} C_DIS
LIN {X -5.9235,Y -4.6928,Z 4,A -3.2389,B 0,C 0,E1 0.1598,E2 90.0709} C_DIS
LIN {X -6.5676,Y -3.7312,Z 4,A -3.2219,B 0,C 0,E1 0.1598,E2 90.0708} C_DIS
LIN {X -7.0494,Y -2.7246,Z 4,A -3.1972,B 0,C 0,E1 0.1598,E2 90.0708} C_DIS
LIN {X -7.3621,Y -1.6865,Z 4,A -3.165,B 0,C 0,E1 0.1598,E2 90.0708} C_DIS
LIN {X -7.5391,Y -0.5182,Z 4,A -3.1222,B 0,C 0,E1 0.1598,E2 90.0708} C_DIS
LIN {X -7.528,Y 0.6121,Z 4,A -3.0742,B 0,C 0,E1 0.1598,E2 90.0708} C_DIS
LIN {X -7.4174,Y 1.4227,Z 4,A -3.0364,B 0,C 0,E1 0.1598,E2 90.0712} C_DIS
LIN {X -7.1188,Y 2.5357,Z 4,A -2.9784,B 0,C 0,E1 0.1598,E2 90.071} C_DIS
LIN {X -6.6343,Y 3.6176,Z 4,A -2.915,B 0,C 0,E1 0.1598,E2 90.0711} C_DIS
LIN {X -6.0252,Y 4.5607,Z 4,A -2.853,B 0,C 0,E1 0.1598,E2 90.0713} C_DIS
LIN {X -5.1879,Y 5.4942,Z 4,A -2.7829,B 0,C 0,E1 0.1598,E2 90.0714} C_DIS
LIN {X -4.2752,Y 6.2308,Z 4,A -2.7184,B 0,C 0,E1 0.1598,E2 90.0717} C_DIS
LIN {X -3.4635,Y 6.717,Z 4,A -2.6681,B 0,C 0,E1 0.1598,E2 90.0719} C_DIS
LIN {X -2.3551,Y 7.181,Z 4,A -2.6077,B 0,C 0,E1 0.1598,E2 90.072} C_DIS
LIN {X -0.278,Y 7.5526,Z 4,A -2.5154,B 0,C 0,E1 0.1598,E2 90.0722} C_DIS
LIN {X 0.7269,Y 7.5229,Z 4,A -2.4796,B 0,C 0,E1 0.1598,E2 90.0722} C_DIS
LIN {X 1.9985,Y 7.2883,Z 4,A -2.4425,B 0,C 0,E1 0.1598,E2 90.0722} C_DIS
LIN {X 3.2756,Y 6.8097,Z 4,A -2.4155,B 0,C 0,E1 0.1598,E2 90.0722} C_DIS
LIN {X 4.4658,Y 6.0905,Z 4,A -2.4018,B 0,C 0,E1 0.1598,E2 90.072} C_DIS
LIN {X 5.1438,Y 5.5296,Z 4,A -2.4006,B 0,C 0,E1 0.1598,E2 90.0722} C_DIS
LIN {X 6.0394,Y 4.5407,Z 4,A -2.4091,B 0,C 0,E1 0.1598,E2 90.0718} C_DIS
LIN {X 6.5514,Y 3.7684,Z 4,A -2.4231,B 0,C 0,E1 0.1598,E2 90.0719} C_DIS
LIN {X 7.0315,Y 2.7719,Z 4,A -2.4475,B 0,C 0,E1 0.1598,E2 90.0719} C_DIS
LIN {X 7.3678,Y 1.6846,Z 4,A -2.481,B 0,C 0,E1 0.1598,E2 90.0716} C_DIS
LIN {X 7.5324,Y 0.6177,Z 4,A -2.5202,B 0,C 0,E1 0.1598,E2 90.0716} C_DIS
LIN {X 7.5522,Y -0.2967,Z 4,A -2.5585,B 0,C 0,E1 0.1598,E2 90.0717} C_DIS
LIN {X 7.3908,Y -1.5624,Z 4,A -2.6176,B 0,C 0,E1 0.1598,E2 90.0712} C_DIS
LIN {X 7.0481,Y -2.7282,Z 4,A -2.6799,B 0,C 0,E1 0.1598,E2 90.0713} C_DIS
LIN {X 6.6303,Y -3.6159,Z 4,A -2.7332,B 0,C 0,E1 0.1598,E2 90.0715} C_DIS
LIN {X 6.2191,Y -4.2844,Z 4,A -2.7768,B 0,C 0,E1 0.1598,E2 90.0716} C_DIS
LIN {X 5.7404,Y -4.9063,Z 4,A -2.8208,B 0,C 0,E1 0.1598,E2 90.0716} C_DIS
LIN {X 5.2016,Y -5.4769,Z 4,A -2.8648,B 0,C 0,E1 0.1598,E2 90.0716} C_DIS
LIN {X 4.4511,Y -6.109,Z 4,A -2.9191,B 0,C 0,E1 0.1598,E2 90.0715} C_DIS
LIN {X 3.4599,Y -6.7137,Z 4,A -2.9812,B 0,C 0,E1 0.1598,E2 90.0715} C_DIS
LIN {X 2.3463,Y -7.1838,Z 4,A -3.042,B 0,C 0,E1 0.1598,E2 90.0715} C_DIS
LIN {X 1.4905,Y -7.4085,Z 4,A -3.083,B 0,C 0,E1 0.1598,E2 90.0715} C_DIS
LIN {X 0.4602,Y -7.5412,Z 4,A -3.1264,B 0,C 0,E1 0.1598,E2 90.0715} C_DIS
LIN {X 0.4602,Y -7.5412,Z 4,A -3.1264,B 0,C 0,E1 0.1598,E2 90.0715} C_DIS
Enddeposition()
LIN {X -0.0489,Y -8.4894,Z 4,A -3.1843,B 0,C 0,E1 0.1598,E2 90.0702} C_DIS
Startdeposition()
$VEL.CP = VEL_PRINT
LIN {X 0.9831,Y -8.4334,Z 4,A -3.1451,B 0,C 0,E1 0.1598,E2 90.0713} C_DIS
LIN {X 2.1496,Y -8.2111,Z 4,A -3.093,B 0,C 0,E1 0.1598,E2 90.0714} C_DIS
LIN {X 2.9712,Y -7.9488,Z 4,A -3.0518,B 0,C 0,E1 0.1598,E2 90.0714} C_DIS
LIN {X 3.7629,Y -7.6068,Z 4,A -3.0082,B 0,C 0,E1 0.1598,E2 90.0715} C_DIS
LIN {X 4.5158,Y -7.186,Z 4,A -2.9627,B 0,C 0,E1 0.1598,E2 90.0715} C_DIS
LIN {X 5.2223,Y -6.6913,Z 4,A -2.9158,B 0,C 0,E1 0.1598,E2 90.0715} C_DIS
LIN {X 6.0914,Y -5.9148,Z 4,A -2.8508,B 0,C 0,E1 0.1598,E2 90.0715} C_DIS
LIN {X 6.7556,Y -5.1387,Z 4,A -2.7934,B 0,C 0,E1 0.1598,E2 90.0715} C_DIS
LIN {X 7.2182,Y -4.465,Z 4,A -2.7479,B 0,C 0,E1 0.1598,E2 90.0717} C_DIS
LIN {X 7.6142,Y -3.75,Z 4,A -2.703,B 0,C 0,E1 0.1598,E2 90.0717} C_DIS
LIN {X 7.9398,Y -3.0003,Z 4,A -2.6591,B 0,C 0,E1 0.1598,E2 90.0717} C_DIS
LIN {X 8.192,Y -2.2228,Z 4,A -2.6168,B 0,C 0,E1 0.1598,E2 90.0717} C_DIS
LIN {X 8.4206,Y -1.0955,Z 4,A -2.5602,B 0,C 0,E1 0.1598,E2 90.0715} C_DIS
LIN {X 8.4872,Y -0.1108,Z 4,A -2.5161,B 0,C 0,E1 0.1598,E2 90.0717} C_DIS
LIN {X 8.461,Y 0.6783,Z 4,A -2.4837,B 0,C 0,E1 0.1598,E2 90.0719} C_DIS
LIN {X 8.3277,Y 1.6564,Z 4,A -2.4469,B 0,C 0,E1 0.1598,E2 90.0717} C_DIS
LIN {X 8.0121,Y 2.7956,Z 4,A -2.4101,B 0,C 0,E1 0.1598,E2 90.0717} C_DIS
LIN {X 7.7085,Y 3.5486,Z 4,A -2.3897,B 0,C 0,E1 0.1598,E2 90.072} C_DIS
LIN {X 7.3344,Y 4.2693,Z 4,A -2.373,B 0,C 0,E1 0.1598,E2 90.0721} C_DIS
LIN {X 6.8935,Y 4.9512,Z 4,A -2.3604,B 0,C 0,E1 0.1598,E2 90.0721} C_DIS
LIN {X 6.3896,Y 5.588,Z 4,A -2.3521,B 0,C 0,E1 0.1598,E2 90.0721} C_DIS
LIN {X 5.8271,Y 6.1737,Z 4,A -2.3481,B 0,C 0,E1 0.1598,E2 90.0722} C_DIS
LIN {X 4.9633,Y 6.8901,Z 4,A -2.3496,B 0,C 0,E1 0.1598,E2 90.0722} C_DIS
LIN {X 4.0831,Y 7.4413,Z 4,A -2.3589,B 0,C 0,E1 0.1598,E2 90.0722} C_DIS
LIN {X 3.3359,Y 7.8047,Z 4,A -2.3712,B 0,C 0,E1 0.1598,E2 90.0723} C_DIS
LIN {X 2.5566,Y 8.0929,Z 4,A -2.3878,B 0,C 0,E1 0.1598,E2 90.0723} C_DIS
LIN {X 1.7532,Y 8.3045,Z 4,A -2.4086,B 0,C 0,E1 0.1598,E2 90.0723} C_DIS
LIN {X 0.9329,Y 8.4367,Z 4,A -2.4333,B 0,C 0,E1 0.1598,E2 90.0723} C_DIS
LIN {X 0.1036,Y 8.4875,Z 4,A -2.4618,B 0,C 0,E1 0.1598,E2 90.0723} C_DIS
LIN {X -0.7266,Y 8.4559,Z 4,A -2.4938,B 0,C 0,E1 0.1598,E2 90.0723} C_DIS
LIN {X -1.5498,Y 8.3438,Z 4,A -2.529,B 0,C 0,E1 0.1598,E2 90.0722} C_DIS
LIN {X -2.3582,Y 8.1521,Z 4,A -2.5669,B 0,C 0,E1 0.1598,E2 90.0722} C_DIS
LIN {X -3.144,Y 7.8823,Z 4,A -2.6072,B 0,C 0,E1 0.1598,E2 90.0721} C_DIS
LIN {X -3.8997,Y 7.5372,Z 4,A -2.6496,B 0,C 0,E1 0.1598,E2 90.072} C_DIS
LIN {X -4.6183,Y 7.1201,Z 4,A -2.6937,B 0,C 0,E1 0.1598,E2 90.0719} C_DIS
LIN {X -5.2927,Y 6.6349,Z 4,A -2.7389,B 0,C 0,E1 0.1598,E2 90.0719} C_DIS
LIN {X -5.9167,Y 6.0862,Z 4,A -2.785,B 0,C 0,E1 0.1598,E2 90.0717} C_DIS
LIN {X -6.4838,Y 5.4789,Z 4,A -2.8314,B 0,C 0,E1 0.1598,E2 90.0717} C_DIS
LIN {X -6.9885,Y 4.8189,Z 4,A -2.8777,B 0,C 0,E1 0.1598,E2 90.0715} C_DIS
LIN {X -7.4261,Y 4.1125,Z 4,A -2.9235,B 0,C 0,E1 0.1598,E2 90.0715} C_DIS
LIN {X -7.7928,Y 3.3668,Z 4,A -2.9683,B 0,C 0,E1 0.1598,E2 90.0713} C_DIS
LIN {X -8.148,Y 2.3908,Z 4,A -3.0221,B 0,C 0,E1 0.1598,E2 90.071} C_DIS
LIN {X -8.3771,Y 1.3741,Z 4,A -3.0733,B 0,C 0,E1 0.1598,E2 90.071} C_DIS
LIN {X -8.4864,Y 0.2801,Z 4,A -3.1232,B 0,C 0,E1 0.1598,E2 90.0708} C_DIS
LIN {X -8.4563,Y -0.7249,Z 4,A -3.1645,B 0,C 0,E1 0.1598,E2 90.0708} C_DIS
LIN {X -8.3494,Y -1.5223,Z 4,A -3.1942,B 0,C 0,E1 0.1598,E2 90.071} C_DIS
LIN {X -8.168,Y -2.3061,Z 4,A -3.2205,B 0,C 0,E1 0.1598,E2 90.071} C_DIS
LIN {X -7.9134,Y -3.0692,Z 4,A -3.2433,B 0,C 0,E1 0.1598,E2 90.071} C_DIS
LIN {X -7.587,Y -3.8047,Z 4,A -3.2623,B 0,C 0,E1 0.1598,E2 90.071} C_DIS
LIN {X -7.1925,Y -4.5058,Z 4,A -3.2773,B 0,C 0,E1 0.1598,E2 90.071} C_DIS
LIN {X -6.6129,Y -5.3276,Z 4,A -3.2905,B 0,C 0,E1 0.1598,E2 90.0708} C_DIS
LIN {X -5.7805,Y -6.2155,Z 4,A -3.2974,B 0,C 0,E1 0.1598,E2 90.0708} C_DIS
LIN {X -5.1588,Y -6.7407,Z 4,A -3.297,B 0,C 0,E1 0.1598,E2 90.071} C_DIS
LIN {X -4.4896,Y -7.2038,Z 4,A -3.292,B 0,C 0,E1 0.1598,E2 90.071} C_DIS
LIN {X -3.779,Y -7.6007,Z 4,A -3.2827,B 0,C 0,E1 0.1598,E2 90.0711} C_DIS
LIN {X -3.0335,Y -7.9276,Z 4,A -3.2692,B 0,C 0,E1 0.1598,E2 90.0711} C_DIS
LIN {X -2.2601,Y -8.1811,Z 4,A -3.2516,B 0,C 0,E1 0.1598,E2 90.0712} C_DIS
LIN {X -1.4663,Y -8.3602,Z 4,A -3.2301,B 0,C 0,E1 0.1598,E2 90.0712} C_DIS
LIN {X -0.6589,Y -8.4626,Z 4,A -3.2049,B 0,C 0,E1 0.1598,E2 90.0712} C_DIS
LIN {X -0.6589,Y -8.4626,Z 4,A -3.2049,B 0,C 0,E1 0.1598,E2 90.0712} C_DIS
Enddeposition()
LIN {X 0.0002,Y -4.7527,Z 5,A -3.0083,B 0,C 0,E1 0.1598,E2 90.0603} C_DIS
Startdeposition()
$VEL.CP = VEL_PRINT
LIN {X 0.0002,Y -4.7527,Z 5,A -3.014,B 0,C 0,E1 0.1598,E2 90.066} C_DIS
LIN {X -0.816,Y -4.6817,Z 5,A -3.0458,B 0,C 0,E1 0.1598,E2 90.0709} C_DIS
LIN {X -1.4523,Y -4.5236,Z 5,A -3.063,B 0,C 0,E1 0.1598,E2 90.0714} C_DIS
LIN {X -2.0616,Y -4.2814,Z 5,A -3.0752,B 0,C 0,E1 0.1598,E2 90.0714} C_DIS
LIN {X -2.6307,Y -3.9559,Z 5,A -3.0823,B 0,C 0,E1 0.1598,E2 90.0714} C_DIS
LIN {X -3.1502,Y -3.5561,Z 5,A -3.0845,B 0,C 0,E1 0.1598,E2 90.0714} C_DIS
LIN {X -3.6107,Y -3.0898,Z 5,A -3.0817,B 0,C 0,E1 0.1598,E2 90.0714} C_DIS
LIN {X -4.0021,Y -2.5635,Z 5,A -3.0739,B 0,C 0,E1 0.1598,E2 90.0714} C_DIS
LIN {X -4.3154,Y -1.9875,Z 5,A -3.0611,B 0,C 0,E1 0.1598,E2 90.0714} C_DIS
LIN {X -4.5472,Y -1.3743,Z 5,A -3.0437,B 0,C 0,E1 0.1598,E2 90.0714} C_DIS
LIN {X -4.6931,Y -0.7352,Z 5,A -3.0221,B 0,C 0,E1 0.1598,E2 90.0714} C_DIS
LIN {X -4.751,Y -0.0824,Z 5,A -2.9967,B 0,C 0,E1 0.1598,E2 90.0714} C_DIS
LIN {X -4.7182,Y 0.5724,Z 5,A -2.9679,B 0,C 0,E1 0.1598,E2 90.0714} C_DIS
LIN {X -4.5931,Y 1.2162,Z 5,A -2.9362,B 0,C 0,E1 0.1598,E2 90.0714} C_DIS
LIN {X -4.3816,Y 1.8368,Z 5,A -2.9023,B 0,C 0,E1 0.1598,E2 90.0715} C_DIS
LIN {X -4.0868,Y 2.4223,Z 5,A -2.8668,B 0,C 0,E1 0.1598,E2 90.0715} C_DIS
LIN {X -3.7148,Y 2.962,Z 5,A -2.8304,B 0,C 0,E1 0.1598,E2 90.0717} C_DIS
LIN {X -3.2709,Y 3.4444,Z 5,A -2.7937,B 0,C 0,E1 0.1598,E2 90.0717} C_DIS
LIN {X -2.7674,Y 3.8642,Z 5,A -2.7575,B 0,C 0,E1 0.1598,E2 90.0718} C_DIS
LIN {X -2.2082,Y 4.2067,Z 5,A -2.7225,B 0,C 0,E1 0.1598,E2 90.0718} C_DIS
LIN {X -1.6082,Y 4.4708,Z 5,A -2.6893,B 0,C 0,E1 0.1598,E2 90.072} C_DIS
LIN {X -0.9775,Y 4.65,Z 5,A -2.6585,B 0,C 0,E1 0.1598,E2 90.072} C_DIS
LIN {X -0.3282,Y 4.7417,Z 5,A -2.6307,B 0,C 0,E1 0.1598,E2 90.072} C_DIS
LIN {X 0.3276,Y 4.7414,Z 5,A -2.6065,B 0,C 0,E1 0.1598,E2 90.072} C_DIS
LIN {X 0.9769,Y 4.6501,Z 5,A -2.5864,B 0,C 0,E1 0.1598,E2 90.0721} C_DIS
LIN {X 1.6077,Y 4.4712,Z 5,A -2.5707,B 0,C 0,E1 0.1598,E2 90.0721} C_DIS
LIN {X 2.2071,Y 4.2057,Z 5,A -2.5598,B 0,C 0,E1 0.1598,E2 90.0721} C_DIS
LIN {X 2.765,Y 3.8619,Z 5,A -2.5537,B 0,C 0,E1 0.1598,E2 90.0721} C_DIS
LIN {X 3.2724,Y 3.4467,Z 5,A -2.5526,B 0,C 0,E1 0.1598,E2 90.0721} C_DIS
LIN {X 3.7147,Y 2.9627,Z 5,A -2.5567,B 0,C 0,E1 0.1598,E2 90.0721} C_DIS
LIN {X 4.0871,Y 2.4231,Z 5,A -2.5658,B 0,C 0,E1 0.1598,E2 90.072} C_DIS
LIN {X 4.3808,Y 1.8371,Z 5,A -2.5797,B 0,C 0,E1 0.1598,E2 90.072} C_DIS
LIN {X 4.5928,Y 1.2167,Z 5,A -2.5982,B 0,C 0,E1 0.1598,E2 90.0719} C_DIS
LIN {X 4.7178,Y 0.573,Z 5,A -2.6208,B 0,C 0,E1 0.1598,E2 90.0719} C_DIS
LIN {X 4.7508,Y -0.0818,Z 5,A -2.6473,B 0,C 0,E1 0.1598,E2 90.0719} C_DIS
LIN {X 4.6942,Y -0.7349,Z 5,A -2.6771,B 0,C 0,E1 0.1598,E2 90.0718} C_DIS
LIN {X 4.4957,Y -1.5295,Z 5,A -2.7179,B 0,C 0,E1 0.1598,E2 90.0716} C_DIS
LIN {X 4.1671,Y -2.2795,Z 5,A -2.7618,B 0,C 0,E1 0.1598,E2 90.0716} C_DIS
LIN {X 3.8142,Y -2.8318,Z 5,A -2.7983,B 0,C 0,E1 0.1598,E2 90.0716} C_DIS
LIN {X 3.3897,Y -3.3314,Z 5,A -2.8351,B 0,C 0,E1 0.1598,E2 90.0716} C_DIS
LIN {X 2.8316,Y -3.8134,Z 5,A -2.876,B 0,C 0,E1 0.1598,E2 90.0716} C_DIS
LIN {X 2.3523,Y -4.1287,Z 5,A -2.907,B 0,C 0,E1 0.1598,E2 90.0716} C_DIS
LIN {X 1.7616,Y -4.4131,Z 5,A -2.9408,B 0,C 0,E1 0.1598,E2 90.0716} C_DIS
LIN {X 0.9768,Y -4.6475,Z 5,A -2.9795,B 0,C 0,E1 0.1598,E2 90.0716} C_DIS
LIN {X 0.4914,Y -4.7268,Z 5,A -3.0007,B 0,C 0,E1 0.1598,E2 90.0716} C_DIS
LIN {X 0.4914,Y -4.7268,Z 5,A -3.0007,B 0,C 0,E1 0.1598,E2 90.0716} C_DIS
Enddeposition()
LIN {X -0.007,Y -5.6867,Z 5,A -3.0586,B 0,C 0,E1 0.1598,E2 90.0703} C_DIS
Startdeposition()
$VEL.CP = VEL_PRINT
LIN {X 0.9567,Y -5.6088,Z 5,A -3.021,B 0,C 0,E1 0.1598,E2 90.0715} C_DIS
LIN {X 2.0388,Y -5.3067,Z 5,A -2.9685,B 0,C 0,E1 0.1598,E2 90.0715} C_DIS
LIN {X 2.7577,Y -4.9725,Z 5,A -2.928,B 0,C 0,E1 0.1598,E2 90.0716} C_DIS
LIN {X 3.4216,Y -4.5393,Z 5,A -2.8852,B 0,C 0,E1 0.1598,E2 90.0716} C_DIS
LIN {X 4.0191,Y -4.0188,Z 5,A -2.8412,B 0,C 0,E1 0.1598,E2 90.0716} C_DIS
LIN {X 4.5378,Y -3.4197,Z 5,A -2.7967,B 0,C 0,E1 0.1598,E2 90.0716} C_DIS
LIN {X 4.9723,Y -2.7567,Z 5,A -2.7526,B 0,C 0,E1 0.1598,E2 90.0716} C_DIS
LIN {X 5.307,Y -2.0382,Z 5,A -2.7098,B 0,C 0,E1 0.1598,E2 90.0716} C_DIS
LIN {X 5.5401,Y -1.2803,Z 5,A -2.669,B 0,C 0,E1 0.1598,E2 90.0717} C_DIS
LIN {X 5.663,Y -0.4971,Z 5,A -2.6313,B 0,C 0,E1 0.1598,E2 90.0717} C_DIS
LIN {X 5.675,Y 0.2952,Z 5,A -2.5972,B 0,C 0,E1 0.1598,E2 90.0717} C_DIS
LIN {X 5.5794,Y 1.0819,Z 5,A -2.5674,B 0,C 0,E1 0.1598,E2 90.0718} C_DIS
LIN {X 5.3742,Y 1.8473,Z 5,A -2.5426,B 0,C 0,E1 0.1598,E2 90.0718} C_DIS
LIN {X 5.0646,Y 2.5767,Z 5,A -2.5231,B 0,C 0,E1 0.1598,E2 90.0719} C_DIS
LIN {X 4.6587,Y 3.2574,Z 5,A -2.5093,B 0,C 0,E1 0.1598,E2 90.0719} C_DIS
Enddeposition()
END
